Device.Ch[1].Hz_Count:=Device.RX.DI1_Float.tReal;
Device.Ch[2].Hz_Count:=Device.RX.DI2_Float.tReal;
Device.Ch[3].Hz_Count:=Device.RX.DI3_Float.tReal;
Device.Ch[4].Hz_Count:=Device.RX.DI4_Float.tReal;
Device.Ch[5].Hz_Count:=Device.RX.DI5_Float.tReal;
Device.Ch[6].Hz_Count:=Device.RX.DI6_Float.tReal;
Device.Ch[7].Hz_Count:=Device.RX.DI7_Float.tReal;
Device.Ch[8].Hz_Count:=Device.RX.DI8_Float.tReal;

Device.Ch[1].Totaliser:=Device.RX.DI1_Total.tReal;
Device.Ch[2].Totaliser:=Device.RX.DI2_Total.tReal;
Device.Ch[3].Totaliser:=Device.RX.DI3_Total.tReal;
Device.Ch[4].Totaliser:=Device.RX.DI4_Total.tReal;
Device.Ch[5].Totaliser:=Device.RX.DI5_Total.tReal;
Device.Ch[6].Totaliser:=Device.RX.DI6_Total.tReal;
Device.Ch[7].Totaliser:=Device.RX.DI7_Total.tReal;
Device.Ch[8].Totaliser:=Device.RX.DI8_Total.tReal;

Device.Ch[1].Raw:=Device.RX.DI1_DI_8.tByte[1].0;
Device.Ch[2].Raw:=Device.RX.DI1_DI_8.tByte[1].1;
Device.Ch[3].Raw:=Device.RX.DI1_DI_8.tByte[1].2;
Device.Ch[4].Raw:=Device.RX.DI1_DI_8.tByte[1].3;
Device.Ch[5].Raw:=Device.RX.DI1_DI_8.tByte[1].4;
Device.Ch[6].Raw:=Device.RX.DI1_DI_8.tByte[1].5;
Device.Ch[7].Raw:=Device.RX.DI1_DI_8.tByte[1].6;
Device.Ch[8].Raw:=Device.RX.DI1_DI_8.tByte[1].7;





Device.TX.Counter_Reset.8:=Device.Ch[1].Reset_Count;
Device.TX.Totaliser_Reset.8:=Device.Ch[1].Reset_Totaliser;

Device.TX.Counter_Reset.9:=Device.Ch[2].Reset_Count;
Device.TX.Totaliser_Reset.9:=Device.Ch[2].Reset_Totaliser;

Device.TX.Counter_Reset.10:=Device.Ch[3].Reset_Count;
Device.TX.Totaliser_Reset.10:=Device.Ch[3].Reset_Totaliser;

Device.TX.Counter_Reset.11:=Device.Ch[4].Reset_Count;
Device.TX.Totaliser_Reset.11:=Device.Ch[4].Reset_Totaliser;

Device.TX.Counter_Reset.12:=Device.Ch[5].Reset_Count;
Device.TX.Totaliser_Reset.12:=Device.Ch[5].Reset_Totaliser;

Device.TX.Counter_Reset.13:=Device.Ch[6].Reset_Count;
Device.TX.Totaliser_Reset.13:=Device.Ch[6].Reset_Totaliser;

Device.TX.Counter_Reset.14:=Device.Ch[7].Reset_Count;
Device.TX.Totaliser_Reset.14:=Device.Ch[7].Reset_Totaliser;

Device.TX.Counter_Reset.15:=Device.Ch[8].Reset_Count;
Device.TX.Totaliser_Reset.15:=Device.Ch[8].Reset_Totaliser;

END_FUNCTION

// Level_1/Analog_Pump_HMI_Sync
FUNCTION_BLOCK Analog_Pump_HMI_Sync
VAR_INPUT
	Sync:BOOL;
END_VAR
VAR_OUTPUT
	StrStatus:STRING;
	StrMode:String;
END_VAR
VAR
	Buffer:cAnalog_Pump;
	R_Trig_0: R_trig;
	Sync_1: BOOL;
	Sync_2: BOOL;
	PLC_Changes:UINT;
	HMI_Changes:UINT;
	
END_VAR

VAR_IN_OUT
	HMI:cAnalog_Pump;
	Local:cAnalog_Pump;
END_VAR

(* body of a kind this reader does not render *)

END_FUNCTION_BLOCK

// Level_1/Contactor_HMI_Sync_UDFB
FUNCTION_BLOCK Contactor_HMI_Sync_UDFB
VAR_INPUT
	Sync:BOOL;
END_VAR
VAR_OUTPUT
	strMode:STRING;
	strStatus:STRING;
END_VAR
VAR
	Buffer:Burkert.Contactor_DUT;
	R_Trig_0: R_trig;
	Sync_1: BOOL;
	Sync_2: BOOL;
	PLC_Changes:UINT;
	HMI_Changes:UINT;
	
END_VAR

VAR_IN_OUT
	HMI:Burkert.Contactor_DUT;
	Local:Burkert.Contactor_DUT;
END_VAR

(* body of a kind this reader does not render *)

END_FUNCTION_BLOCK

// Level_1/Eaton_VFD_HMI_Sync
FUNCTION_BLOCK Eaton_VFD_HMI_Sync
VAR_INPUT
	Sync:BOOL;
END_VAR
VAR_OUTPUT
	StrStatus:STRING;
	StrMode:String;
END_VAR
VAR
	Buffer:cVFD_Eaton_DUT;
	R_Trig_0: R_trig;
	Sync_1: BOOL;
	Sync_2: BOOL;
	PLC_Changes:UINT;
	HMI_Changes:UINT;
	
END_VAR

VAR_IN_OUT
	HMI:cVFD_Eaton_DUT;
	Local:cVFD_Eaton_DUT;
END_VAR

(* body of a kind this reader does not render *)

END_FUNCTION_BLOCK

// Level_1/M_Pump_HMI_Sync
FUNCTION_BLOCK M_Pump_HMI_Sync
VAR_INPUT
	Sync:BOOL;
END_VAR
VAR_OUTPUT
	StrStatus:STRING;
	StrMode:String;
END_VAR
VAR
	Buffer:cM_Pump;
	R_Trig_0: R_trig;
	Sync_1: BOOL;
	Sync_2: BOOL;
	PLC_Changes:UINT;
	HMI_Changes:UINT;
	
END_VAR

VAR_IN_OUT
	HMI:cM_Pump;
	Local:cM_Pump;
END_VAR

(* body of a kind this reader does not render *)

END_FUNCTION_BLOCK

// Level_2/PID_HMI_Sync_UDFB
FUNCTION_BLOCK PID_HMI_Sync_UDFB
VAR_INPUT
	Sync:BOOL;
END_VAR
VAR_OUTPUT
	strMode:STRING;
	strStatus:STRING;
END_VAR
VAR
	Buffer:cPID_DUT;
	R_Trig_0: R_trig;
	Sync_1: BOOL;
	Sync_2: BOOL;
	PLC_Changes:UINT;
	HMI_Changes:UINT;
	
END_VAR

VAR_IN_OUT
	HMI:cPID_DUT;
	Local:cPID_DUT;
END_VAR

(* body of a kind this reader does not render *)

END_FUNCTION_BLOCK

// Level_3/Brite_HMI_Sync
FUNCTION_BLOCK Brite_HMI_Sync
VAR_INPUT
	Sync:BOOL;
END_VAR
VAR_OUTPUT
END_VAR
VAR
	Buffer:cBrite_DUT;
	R_Trig_0: R_trig;
	Sync_1: BOOL;
	Sync_2: BOOL;
	PLC_Changes:UINT;
	HMI_Changes:UINT;
	
	//PID_0: PID_HMI_Sync_UDFB;
	PID_Match: BOOL;
	Status_Match: BOOL;
	PID_Coompare: UINT;
	Status_Compare: UINT;
END_VAR

VAR_IN_OUT
	HMI:cBrite_DUT;
	Local:cBrite_DUT;
END_VAR

(* body of a kind this reader does not render *)

END_FUNCTION_BLOCK

// Level_3/Fermenter_HMI_Sync
FUNCTION_BLOCK Fermenter_HMI_Sync
VAR_INPUT
	Sync:BOOL;
END_VAR
VAR_OUTPUT
END_VAR
VAR
	Buffer:cFermenter_DUT;
	R_Trig_0: R_trig;
	Sync_1: BOOL;
	Sync_2: BOOL;
	PLC_Changes:UINT;
	HMI_Changes:UINT;
	
	//PID_0: PID_HMI_Sync_UDFB;
	PID_Match: BOOL;
	Status_Match: BOOL;
	PID_Coompare: UINT;
	Status_Compare: UINT;
END_VAR

VAR_IN_OUT
	HMI:cFermenter_DUT;
	Local:cFermenter_DUT;
END_VAR

(* body of a kind this reader does not render *)

END_FUNCTION_BLOCK

// Adam_6050_FB
FUNCTION Adam_6050_FB : BOOL
VAR_INPUT
	HSC_0_Enable:BOOL:=FALSE;
	HSC_0_Reset:BOOL:=FALSE;
	HSC_1_Enable:BOOL:=FALSE;
	HSC_1_Reset:BOOL:=FALSE;
	HSC_2_Enable:BOOL:=FALSE;
	HSC_2_Reset:BOOL:=FALSE;
	HSC_3_Enable:BOOL:=FALSE;
	HSC_3_Reset:BOOL:=FALSE;
	HSC_4_Enable:BOOL:=FALSE;
	HSC_4_Reset:BOOL:=FALSE;
	HSC_5_Enable:BOOL:=FALSE;
	HSC_5_Reset:BOOL:=FALSE;
	HSC_6_Enable:BOOL:=FALSE;
	HSC_6_Reset:BOOL:=FALSE;
	HSC_7_Enable:BOOL:=FALSE;
	HSC_7_Reset:BOOL:=FALSE;
	HSC_8_Enable:BOOL:=FALSE;
	HSC_8_Reset:BOOL:=FALSE;
	HSC_9_Enable:BOOL:=FALSE;
	HSC_9_Reset:BOOL:=FALSE;
	HSC_10_Enable:BOOL:=FALSE;
	HSC_10_Reset:BOOL:=FALSE;
	HSC_11_Enable:BOOL:=FALSE;
	HSC_11_Reset:BOOL:=FALSE;
	
	DO_0:BOOL:=FALSE;
	DO_1:BOOL:=FALSE;
	DO_2:BOOL:=FALSE;
	DO_3:BOOL:=FALSE;
	DO_4:BOOL:=FALSE;
	DO_5:BOOL:=FALSE;
//	DO_6:BOOL;
//	DO_7:BOOL;
	RX_DI_4x300: WORD;
	RX_Counts_4x0: ARRAY[0..11] OF UDINT;
END_VAR
VAR_OUTPUT
	HSC_0:UDINT;
	HSC_1:UDINT;
	HSC_2:UDINT;
	HSC_3:UDINT;
	HSC_4:UDINT;
	HSC_5:UDINT;
	HSC_6:UDINT;
	HSC_7:UDINT;
	HSC_8:UDINT;
	HSC_9:UDINT;
	HSC_10:UDINT;
	HSC_11:UDINT;
	
	DI_0:BOOL;
	DI_1:BOOL;
	DI_2:BOOL;
	DI_3:BOOL;
	DI_4:BOOL;
	DI_5:BOOL;
	DI_6:BOOL;
	DI_7:BOOL;
	DI_8:BOOL;
	DI_9:BOOL;
	DI_10:BOOL;
	DI_11:BOOL;
	
	

	
	
	TX_DO_4x302: WORD;
	TX_Counts_Control_0x32: ARRAY[0..2] OF WORD;
END_VAR
VAR
END_VAR

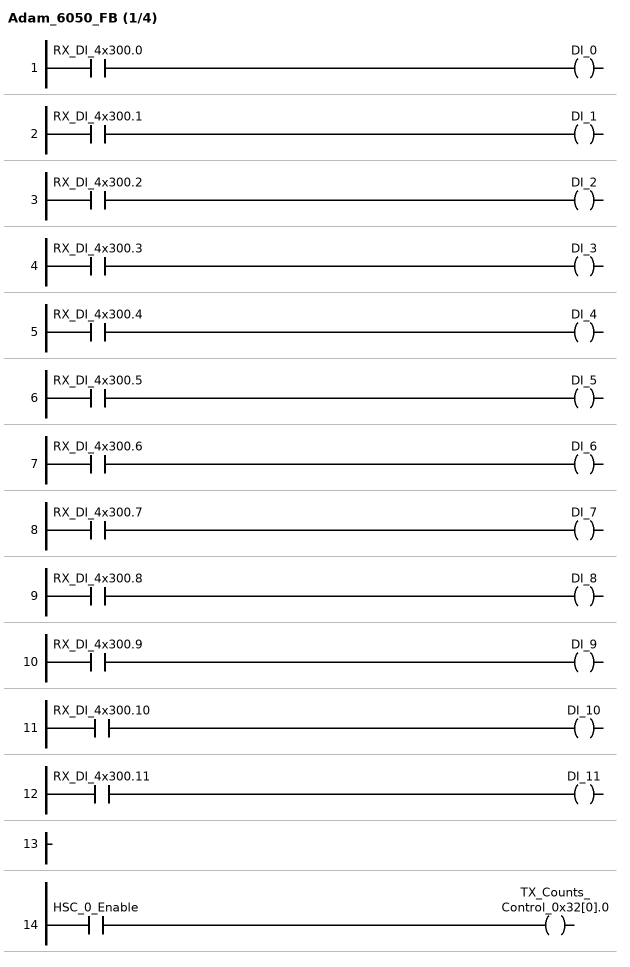
// NETWORK 1
DI_0 := RX_DI_4x300.0;

// NETWORK 2
DI_1 := RX_DI_4x300.1;

// NETWORK 3
DI_2 := RX_DI_4x300.2;

// NETWORK 4
DI_3 := RX_DI_4x300.3;

// NETWORK 5
DI_4 := RX_DI_4x300.4;

// NETWORK 6
DI_5 := RX_DI_4x300.5;

// NETWORK 7
DI_6 := RX_DI_4x300.6;

// NETWORK 8
DI_7 := RX_DI_4x300.7;

// NETWORK 9
DI_8 := RX_DI_4x300.8;

// NETWORK 10
DI_9 := RX_DI_4x300.9;

// NETWORK 11
DI_10 := RX_DI_4x300.10;

// NETWORK 12
DI_11 := RX_DI_4x300.11;

// NETWORK 13

// NETWORK 14
TX_Counts_Control_0x32[0].0 := HSC_0_Enable;

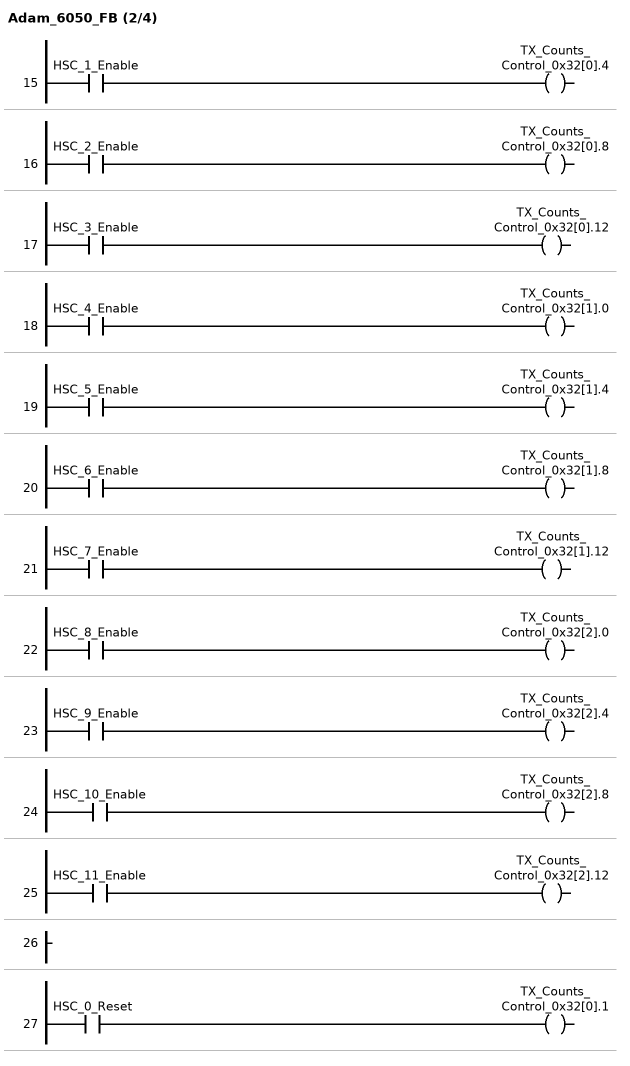
// NETWORK 15
TX_Counts_Control_0x32[0].4 := HSC_1_Enable;

// NETWORK 16
TX_Counts_Control_0x32[0].8 := HSC_2_Enable;

// NETWORK 17
TX_Counts_Control_0x32[0].12 := HSC_3_Enable;

// NETWORK 18
TX_Counts_Control_0x32[1].0 := HSC_4_Enable;

// NETWORK 19
TX_Counts_Control_0x32[1].4 := HSC_5_Enable;

// NETWORK 20
TX_Counts_Control_0x32[1].8 := HSC_6_Enable;

// NETWORK 21
TX_Counts_Control_0x32[1].12 := HSC_7_Enable;

// NETWORK 22
TX_Counts_Control_0x32[2].0 := HSC_8_Enable;

// NETWORK 23
TX_Counts_Control_0x32[2].4 := HSC_9_Enable;

// NETWORK 24
TX_Counts_Control_0x32[2].8 := HSC_10_Enable;

// NETWORK 25
TX_Counts_Control_0x32[2].12 := HSC_11_Enable;

// NETWORK 26

// NETWORK 27
TX_Counts_Control_0x32[0].1 := HSC_0_Reset;

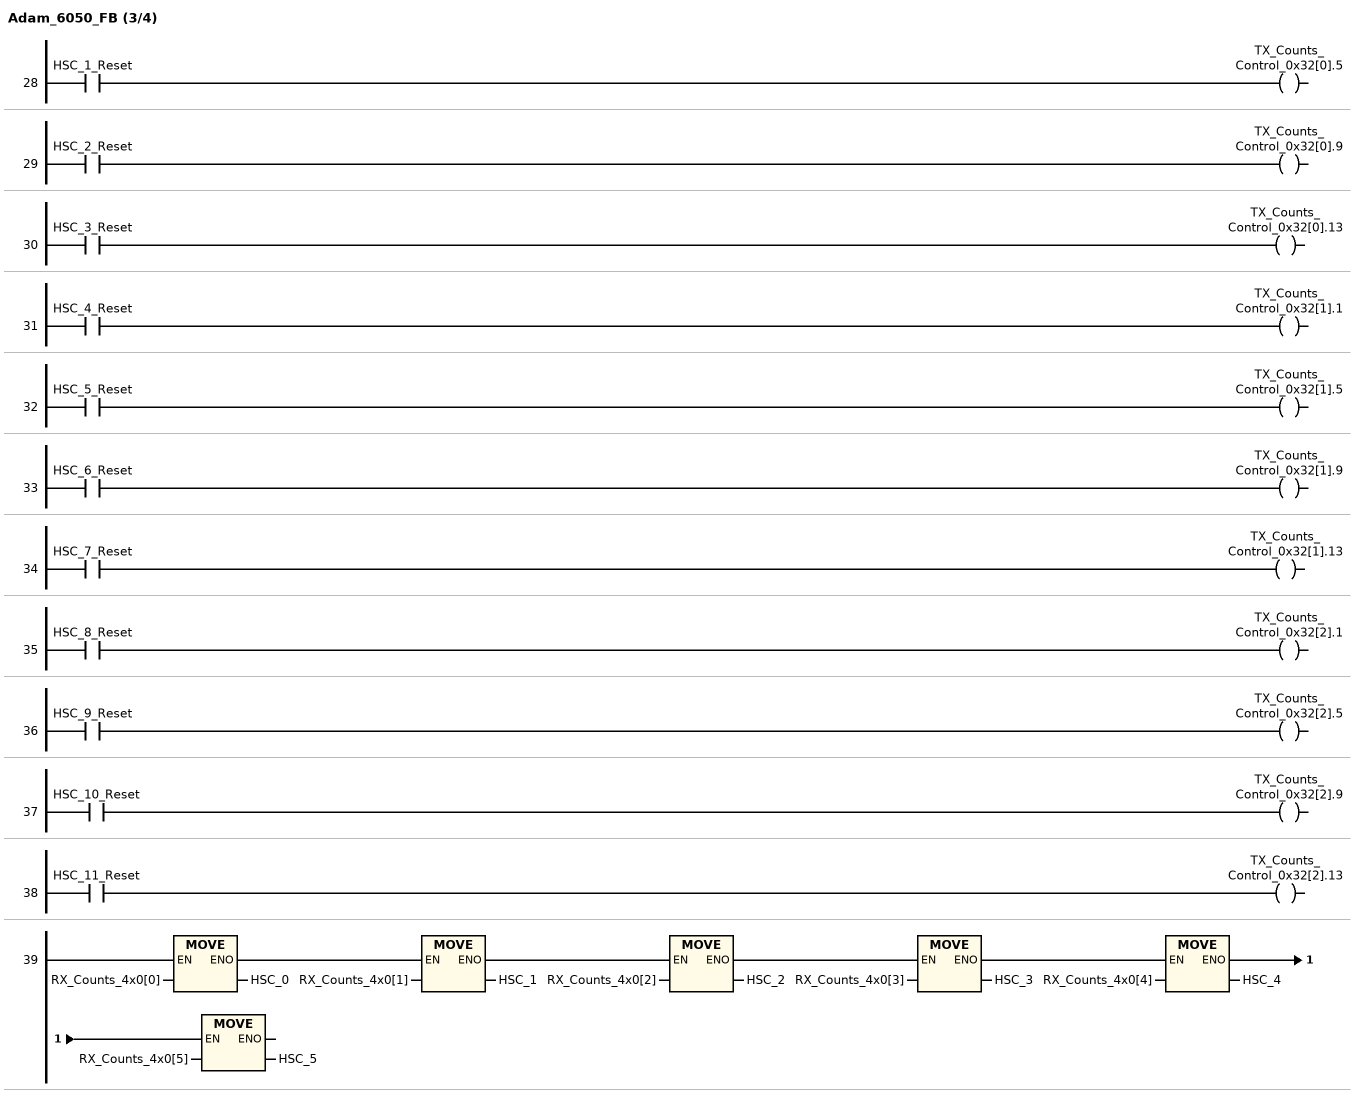
// NETWORK 28
TX_Counts_Control_0x32[0].5 := HSC_1_Reset;

// NETWORK 29
TX_Counts_Control_0x32[0].9 := HSC_2_Reset;

// NETWORK 30
TX_Counts_Control_0x32[0].13 := HSC_3_Reset;

// NETWORK 31
TX_Counts_Control_0x32[1].1 := HSC_4_Reset;

// NETWORK 32
TX_Counts_Control_0x32[1].5 := HSC_5_Reset;

// NETWORK 33
TX_Counts_Control_0x32[1].9 := HSC_6_Reset;

// NETWORK 34
TX_Counts_Control_0x32[1].13 := HSC_7_Reset;

// NETWORK 35
TX_Counts_Control_0x32[2].1 := HSC_8_Reset;

// NETWORK 36
TX_Counts_Control_0x32[2].5 := HSC_9_Reset;

// NETWORK 37
TX_Counts_Control_0x32[2].9 := HSC_10_Reset;

// NETWORK 38
TX_Counts_Control_0x32[2].13 := HSC_11_Reset;

// NETWORK 39
HSC_0 := RX_Counts_4x0[0];
HSC_1 := RX_Counts_4x0[1];
HSC_2 := RX_Counts_4x0[2];
HSC_3 := RX_Counts_4x0[3];
HSC_4 := RX_Counts_4x0[4];
HSC_5 := RX_Counts_4x0[5];

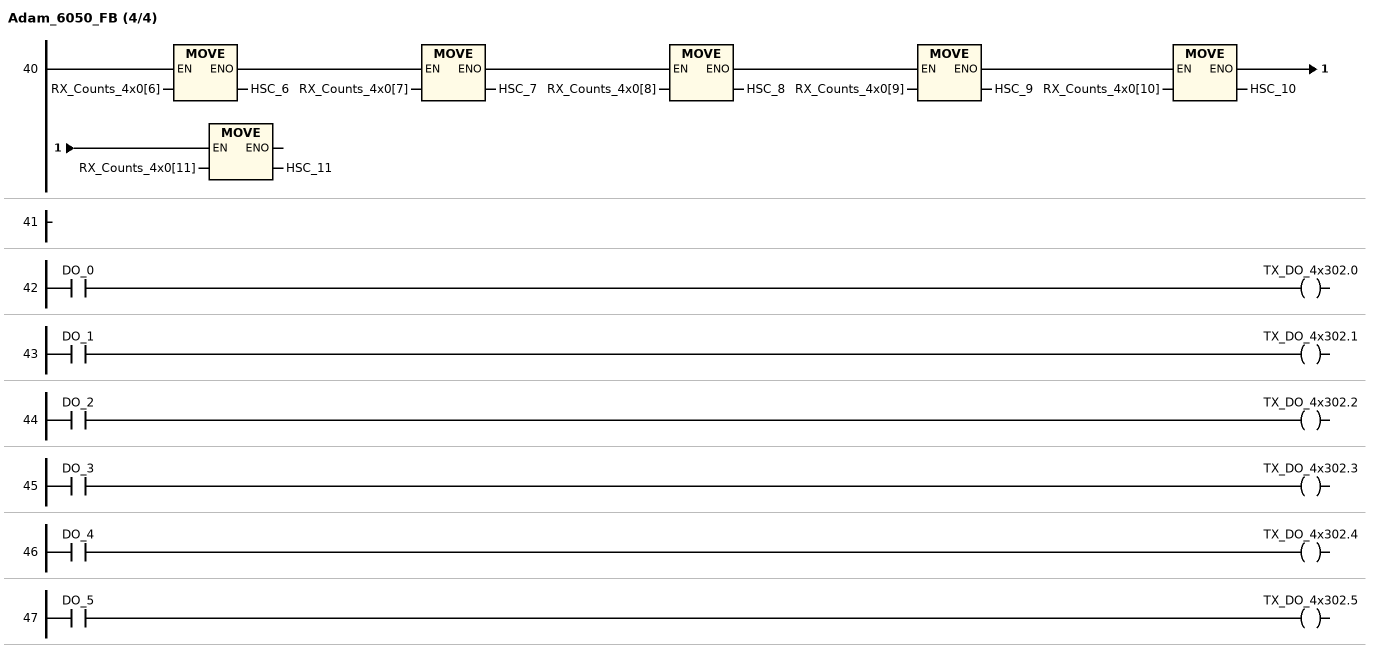
// NETWORK 40
HSC_6 := RX_Counts_4x0[6];
HSC_7 := RX_Counts_4x0[7];
HSC_8 := RX_Counts_4x0[8];
HSC_9 := RX_Counts_4x0[9];
HSC_10 := RX_Counts_4x0[10];
HSC_11 := RX_Counts_4x0[11];

// NETWORK 41

// NETWORK 42
TX_DO_4x302.0 := DO_0;

// NETWORK 43
TX_DO_4x302.1 := DO_1;

// NETWORK 44
TX_DO_4x302.2 := DO_2;

// NETWORK 45
TX_DO_4x302.3 := DO_3;

// NETWORK 46
TX_DO_4x302.4 := DO_4;

// NETWORK 47
TX_DO_4x302.5 := DO_5;

END_FUNCTION

// Adam_6250
FUNCTION Adam_6250 : bool
VAR_INPUT
	Device:REFERENCE TO cAdam_6250;
END_VAR

VAR
END_VAR

Device.DI[0].DI:=Device.Rx_DI.0;
Device.DI[1].DI:=Device.Rx_DI.1;
Device.DI[2].DI:=Device.Rx_DI.2;
Device.DI[3].DI:=Device.Rx_DI.3;
Device.DI[4].DI:=Device.Rx_DI.4;
Device.DI[5].DI:=Device.Rx_DI.5;
Device.DI[6].DI:=Device.Rx_DI.6;
Device.DI[7].DI:=Device.Rx_DI.7;

Device.DI[0].Count:=Device.RX_Counter_Values[0];
Device.DI[1].Count:=Device.RX_Counter_Values[1];
Device.DI[2].Count:=Device.RX_Counter_Values[2];
Device.DI[3].Count:=Device.RX_Counter_Values[3];
Device.DI[4].Count:=Device.RX_Counter_Values[4];
Device.DI[5].Count:=Device.RX_Counter_Values[5];
Device.DI[6].Count:=Device.RX_Counter_Values[6];
Device.DI[7].Count:=Device.RX_Counter_Values[7];

Device.DI[0].Frequency:=TO_REAL(Device.RX_Counter_Values[0])/10;
Device.DI[1].Frequency:=TO_REAL(Device.RX_Counter_Values[1])/10;
Device.DI[2].Frequency:=TO_REAL(Device.RX_Counter_Values[2])/10;
Device.DI[3].Frequency:=TO_REAL(Device.RX_Counter_Values[3])/10;
Device.DI[4].Frequency:=TO_REAL(Device.RX_Counter_Values[4])/10;
Device.DI[5].Frequency:=TO_REAL(Device.RX_Counter_Values[5])/10;
Device.DI[6].Frequency:=TO_REAL(Device.RX_Counter_Values[6])/10;
Device.DI[7].Frequency:=TO_REAL(Device.RX_Counter_Values[7])/10;

Device.Tx_Counter_Control[0].0:=Device.DI[0].Enable_HSC;
Device.Tx_Counter_Control[0].1:=Device.DI[1].Enable_HSC;
Device.Tx_Counter_Control[0].2:=Device.DI[2].Enable_HSC;
Device.Tx_Counter_Control[0].3:=Device.DI[3].Enable_HSC;
Device.Tx_Counter_Control[0].4:=Device.DI[4].Enable_HSC;
Device.Tx_Counter_Control[0].5:=Device.DI[5].Enable_HSC;
Device.Tx_Counter_Control[0].6:=Device.DI[6].Enable_HSC;
Device.Tx_Counter_Control[0].7:=Device.DI[7].Enable_HSC;

Device.Tx_Counter_Control[1].0:=Device.DI[0].Clear_HSC;
Device.Tx_Counter_Control[1].1:=Device.DI[1].Clear_HSC;
Device.Tx_Counter_Control[1].2:=Device.DI[2].Clear_HSC;
Device.Tx_Counter_Control[1].3:=Device.DI[3].Clear_HSC;
Device.Tx_Counter_Control[1].4:=Device.DI[4].Clear_HSC;
Device.Tx_Counter_Control[1].5:=Device.DI[5].Clear_HSC;
Device.Tx_Counter_Control[1].6:=Device.DI[6].Clear_HSC;
Device.Tx_Counter_Control[1].7:=Device.DI[7].Clear_HSC;

Device.Tx_Counter_Control[2].0:=Device.DI[0].Clear_Overflow;
Device.Tx_Counter_Control[2].1:=Device.DI[1].Clear_Overflow;
Device.Tx_Counter_Control[2].2:=Device.DI[2].Clear_Overflow;
Device.Tx_Counter_Control[2].3:=Device.DI[3].Clear_Overflow;
Device.Tx_Counter_Control[2].4:=Device.DI[4].Clear_Overflow;
Device.Tx_Counter_Control[2].5:=Device.DI[5].Clear_Overflow;
Device.Tx_Counter_Control[2].6:=Device.DI[6].Clear_Overflow;
Device.Tx_Counter_Control[2].7:=Device.DI[7].Clear_Overflow;

Device.Tx_DO.0	:=device.Dout[0].Dout;
Device.Tx_DO.1	:=device.Dout[1].Dout;
Device.Tx_DO.2	:=device.Dout[2].Dout;
Device.Tx_DO.3	:=device.Dout[3].Dout;
Device.Tx_DO.4	:=device.Dout[4].Dout;
Device.Tx_DO.5	:=device.Dout[5].Dout;
Device.Tx_DO.6	:=device.Dout[6].Dout;

Device.Tx_Pulse_Width_Low[0] :=Device.Dout[0].Pulse_Output_Low_Width;
Device.Tx_Pulse_Width_Low[1] :=Device.Dout[1].Pulse_Output_Low_Width;
Device.Tx_Pulse_Width_Low[2] :=Device.Dout[2].Pulse_Output_Low_Width;
Device.Tx_Pulse_Width_Low[3] :=Device.Dout[3].Pulse_Output_Low_Width;
Device.Tx_Pulse_Width_Low[4] :=Device.Dout[4].Pulse_Output_Low_Width;
Device.Tx_Pulse_Width_Low[5] :=Device.Dout[5].Pulse_Output_Low_Width;
Device.Tx_Pulse_Width_Low[6] :=Device.Dout[6].Pulse_Output_Low_Width;

Device.Tx_Pulse_Width_High[0]	:=Device.Dout[0].Pulse_Output_High_Width;
Device.Tx_Pulse_Width_High[1]	:=Device.Dout[1].Pulse_Output_High_Width;
Device.Tx_Pulse_Width_High[2]	:=Device.Dout[2].Pulse_Output_High_Width;
Device.Tx_Pulse_Width_High[3]	:=Device.Dout[3].Pulse_Output_High_Width;
Device.Tx_Pulse_Width_High[4]	:=Device.Dout[4].Pulse_Output_High_Width;
Device.Tx_Pulse_Width_High[5]	:=Device.Dout[5].Pulse_Output_High_Width;
Device.Tx_Pulse_Width_High[6]	:=Device.Dout[6].Pulse_Output_High_Width;

Device.Tx_Set_Absolute_Pulse[0]	:=Device.Dout[0].Set_Absolute_Pulse;
Device.Tx_Set_Absolute_Pulse[1]	:=Device.Dout[1].Set_Absolute_Pulse;
Device.Tx_Set_Absolute_Pulse[2]	:=Device.Dout[2].Set_Absolute_Pulse;
Device.Tx_Set_Absolute_Pulse[3]	:=Device.Dout[3].Set_Absolute_Pulse;
Device.Tx_Set_Absolute_Pulse[4]	:=Device.Dout[4].Set_Absolute_Pulse;
Device.Tx_Set_Absolute_Pulse[5]	:=Device.Dout[5].Set_Absolute_Pulse;
Device.Tx_Set_Absolute_Pulse[6]	:=Device.Dout[6].Set_Absolute_Pulse;

Device.Tx_Set_Incremental_Pulse[0]	:=Device.Dout[0].Set_Incremental_Pulse;
Device.Tx_Set_Incremental_Pulse[1]	:=Device.Dout[1].Set_Incremental_Pulse;
Device.Tx_Set_Incremental_Pulse[2]	:=Device.Dout[2].Set_Incremental_Pulse;
Device.Tx_Set_Incremental_Pulse[3]	:=Device.Dout[3].Set_Incremental_Pulse;
Device.Tx_Set_Incremental_Pulse[4]	:=Device.Dout[4].Set_Incremental_Pulse;
Device.Tx_Set_Incremental_Pulse[5]	:=Device.Dout[5].Set_Incremental_Pulse;
Device.Tx_Set_Incremental_Pulse[6]	:=Device.Dout[6].Set_Incremental_Pulse;

END_FUNCTION

// Level_0_Remote_IO/MicroControl/MC4AI
FUNCTION MC4AI 
VAR_INPUT
	GW_TCP_State:ModbusTCPComState;
END_VAR

VAR
END_VAR


VAR_IN_OUT
	GW:MicroControl_4AI;
END_VAR

GW.GW_TCP_State:=GW_TCP_State;

IF NOT(GW_TCP_State=10) THEN
	GW.PV[0]:= (TO_REAL(GW.PV_RX[0])/1000);
	GW.PV[1]:= (TO_REAL(GW.PV_RX[1])/1000);
	GW.PV[2]:= (TO_REAL(GW.PV_RX[2])/1000);
	GW.PV[3]:= (TO_REAL(GW.PV_RX[3])/1000);
ELSE
	GW.PV[0]:=(-9999999);
	GW.PV[1]:=(-9999999);
	GW.PV[2]:=(-9999999);
	GW.PV[3]:=(-9999999);
END_IF;

END_FUNCTION

// MB0_RTD
FUNCTION_BLOCK MB0_RTD
VAR_INPUT
	Online:BOOL;
	Device: REFERENCE TO cMB0_RTD;
	
	CH1: REFERENCE TO 	Burkert.cAIT;
	CH1_Probe_Type:		eMB0_RTD_Input_Type;
	CH2: REFERENCE TO 	Burkert.cAIT;
	CH2_Probe_Type:		eMB0_RTD_Input_Type;
	CH3: REFERENCE TO 	Burkert.cAIT;
	CH3_Probe_Type:		eMB0_RTD_Input_Type;
	CH4: REFERENCE TO 	Burkert.cAIT;
	CH4_Probe_Type:		eMB0_RTD_Input_Type;
	System_Units:eUnits;
END_VAR
VAR_OUTPUT
END_VAR
VAR
	Alarm:ARRAY[0..3] OF Burkert.Analog_Alarm_UDFB;
END_VAR

CASE System_Units OF
	eUnits.C:
		Device.TX.Holding_1218[0]:=eMB0_RTD_Units.C;
		Device.TX.Holding_1218[1]:=eMB0_RTD_Units.C;
		Device.TX.Holding_1218[2]:=eMB0_RTD_Units.C;
		Device.TX.Holding_1218[3]:=eMB0_RTD_Units.C;
	eUnits.F:
		Device.TX.Holding_1218[0]:=eMB0_RTD_Units.F;
		Device.TX.Holding_1218[1]:=eMB0_RTD_Units.F;
		Device.TX.Holding_1218[2]:=eMB0_RTD_Units.F;
		Device.TX.Holding_1218[3]:=eMB0_RTD_Units.F;
	eUnits.K:
		Device.TX.Holding_1218[0]:=eMB0_RTD_Units.k;
		Device.TX.Holding_1218[1]:=eMB0_RTD_Units.k;
		Device.TX.Holding_1218[2]:=eMB0_RTD_Units.k;
		Device.TX.Holding_1218[3]:=eMB0_RTD_Units.k;
END_CASE

Device.TX.Holding_31[0]:=CH1_Probe_Type;
Device.TX.Holding_31[1]:=CH1_Probe_Type;
Device.TX.Holding_31[2]:=CH1_Probe_Type;
Device.TX.Holding_31[3]:=CH1_Probe_Type;


CH1.Sensor.EU:=TO_REAL(Device.RX.Holding_41[0])/10;
CH2.Sensor.EU:=TO_REAL(Device.RX.Holding_41[1])/10;
CH3.Sensor.EU:=TO_REAL(Device.RX.Holding_41[2])/10;
CH4.Sensor.EU:=TO_REAL(Device.RX.Holding_41[3])/10;

Alarm[0](
	Config:=CH1.Sensor.Alarm_Config,
	EU:=CH1.Sensor.EU,
	Debounce_Active:=CH1.Sensor.Alarm_Config.Silence, 
	Status =>CH1.Sensor.Status.eStatus,
	Percent_Alarm=>CH1.Sensor.Alarm_Config.PCT_Alarm
	);
Alarm[1](
	Config:=CH2.Sensor.Alarm_Config,
	EU:=CH2.Sensor.EU,
	Debounce_Active:=CH2.Sensor.Alarm_Config.Silence, 
	Status =>CH2.Sensor.Status.eStatus,
	Percent_Alarm=>CH2.Sensor.Alarm_Config.PCT_Alarm
	);
Alarm[2](
	Config:=CH3.Sensor.Alarm_Config,
	EU:=CH3.Sensor.EU,
	Debounce_Active:=CH3.Sensor.Alarm_Config.Silence, 
	Status =>CH3.Sensor.Status.eStatus,
	Percent_Alarm=>CH3.Sensor.Alarm_Config.PCT_Alarm
	);
Alarm[3](
	Config:=CH4.Sensor.Alarm_Config,
	EU:=CH4.Sensor.EU,
	Debounce_Active:=CH4.Sensor.Alarm_Config.Silence, 
	Status =>CH4.Sensor.Status.eStatus,
	Percent_Alarm=>CH4.Sensor.Alarm_Config.PCT_Alarm
	);
	
IF NOT(Online) THEN
	CH1.Sensor.Status.eStatus:=Burkert.eSensor_Status.Offline;
	CH2.Sensor.Status.eStatus:=Burkert.eSensor_Status.Offline;
	CH3.Sensor.Status.eStatus:=Burkert.eSensor_Status.Offline;
	CH4.Sensor.Status.eStatus:=Burkert.eSensor_Status.Offline;
END_IF

END_FUNCTION_BLOCK

// Level_1_Devices/Burkert Library/Analog_Alarm_UDFB
FUNCTION_BLOCK Analog_Alarm_UDFB
VAR_INPUT
	Config	:	REFERENCE TO Burkert.cAlarm_Config;
	EU:REAL  ;
	Debounce_Active:BOOL;
	
END_VAR
VAR_OUTPUT
	Status:eSensor_Status;
	Percent_Alarm:REAL;
	
END_VAR
VAR
	ALARM: BURKERT_OSCAT_BASIC.ALARM_2;
	Warn_Debounce: TON;
	Alarm_Debounce: TON;
	ALarm_PCT:ARRAY[0..4] OF REAL;
	
END_VAR

Status:=run();

METHOD run : eSensor_Status
VAR_INPUT

END_VAR

VAR_OUTPUT

END_VAR
(* body of a kind this reader does not render *)
END_METHOD

END_FUNCTION_BLOCK

// SIO_MB12CDR
FUNCTION_BLOCK SIO_MB12CDR
VAR_INPUT
	Online:BOOL;
	Device : REFERENCE TO cSIO_MB12CDR;
	FIT_0:REFERENCE TO Burkert.cBase_FIT;
	FIT_1:REFERENCE TO Burkert.cBase_FIT;
	FIT_2:REFERENCE TO	Burkert.cBase_FIT;
	FIT_3:REFERENCE TO Burkert.cBase_FIT;
END_VAR
VAR_OUTPUT
END_VAR
VAR
END_VAR

END_FUNCTION_BLOCK

// Contactor
FUNCTION_BLOCK Contactor
VAR_INPUT
	NO_OL:BOOL;
	NO_FWD_Aux:BOOL;
	NO_REV_Aux:BOOL;


	Allow_Reverse:BOOL;
	Inhibit_FWD:BOOL:=FALSE;
	Inhibit_Rev:BOOL:=FALSE;
	Bump_Duration:TIME:=T#1S;
END_VAR

VAR_IN_OUT
	Contactor:cContactor;
END_VAR

VAR_OUTPUT
	Q_FWD:BOOL;
	Q_REV:Bool;
END_VAR


VAR
	local_FWD:BOOL;
	Local_Rev:BOOL;
	Bump_Timer:TP;
	Engage_Ton:TON;
	
END_VAR

Bump_Timer(
	PT:=Bump_Duration, 
	IN:= (Contactor.Mode.eMode=Contactor_modes.Bump_FWD OR Contactor.Mode.eMode=Contactor_modes.Bump_rev)
);
	

Engage_Ton(PT:=T#1S, IN:=(Q_FWD OR Q_REV));

CASE Contactor.Mode.eMode OF
	Contactor_modes.Disabled:
		Local_FWD:=FALSE;
		Local_Rev:=FALSE;
	Contactor_modes.Auto:
		Local_FWD:=Contactor.PLC_CMD_FWD;
		Local_Rev:=Contactor.PLC_CMD_Rev;
	Contactor_modes.Bump_FWD:
		Local_FWD:=Bump_Timer.Q;
		Local_REV:=FALSE;
	Contactor_modes.Bump_REV:
		Local_FWD:=FALSE;
		Local_REV:=Bump_Timer.Q;
	Contactor_modes.Fwd:
		Local_FWD:=TRUE;
		Local_Rev:=FALSE;
	Contactor_modes.Rev:
		Local_FWD:=FALSE;
		Local_Rev:=TRUE;
END_CASE

//IF Inhibit_FWD THEN local_FWD:=FALSE; END_IF;
//IF Inhibit_Rev THEN Local_REv:=FALSE;	END_IF;
IF NO_OL	THEN 
	Local_FWD:=FALSE;
	Local_Rev:=FALSE;
END_IF;

IF (Local_FWD AND Local_REV) THEN
	Local_FWD:=FALSE;
	Local_Rev:=FALSE;
END_IF;

Q_FWD:=Local_FWD AND NOT(Inhibit_FWD);
Q_Rev:=Local_Rev AND NOT(Inhibit_Rev);

Status();

ACTION Status:
Contactor.Ready :=(
	Contactor.Mode.eMode=Contactor_modes.Auto AND
	NOT(NO_OL)
);

Contactor.Status.eStatus:=eContactor_Status.Idle;
IF Contactor.Mode.eMode=Contactor_modes.Disabled THEN	Contactor.Status.eStatus:=eContactor_Status.Disabled; END_IF;




IF Contactor.Mode.eMode=Contactor_modes.Auto AND Contactor.PLC_CMD_FWD THEN Contactor.Status.eStatus:=eContactor_Status.Auto_FWD; END_IF;
IF Contactor.Mode.eMode=Contactor_modes.Auto AND Contactor.PLC_CMD_REV THEN Contactor.Status.eStatus:=eContactor_Status.Auto_Rev; END_IF;

IF Contactor.Mode.eMode=Contactor_modes.Bump_FWD AND Bump_Timer.Q THEN Contactor.Status.eStatus:=eContactor_Status.Manual_FWD; END_IF;
IF Contactor.Mode.eMode=Contactor_modes.Bump_Rev AND Bump_Timer.Q THEN Contactor.Status.eStatus:=eContactor_Status.Manual_REV; END_IF;

IF Contactor.Mode.eMode=Contactor_modes.Fwd  THEN Contactor.Status.eStatus:=eContactor_Status.Manual_FWD; END_IF;
IF Contactor.Mode.eMode=Contactor_modes.rev  THEN Contactor.Status.eStatus:=eContactor_Status.Manual_REV; END_IF;


IF Local_FWD AND NO_FWD_Aux THEN	Contactor.Status.eStatus:=eContactor_Status.FWD_Limit; END_IF;
IF Local_Rev AND NO_Rev_Aux THEN	Contactor.Status.eStatus:=eContactor_Status.Rev_Limit; END_IF;

IF Engage_Ton.Q AND NOT(NO_FWD_Aux OR NO_REV_Aux) THEN Contactor.Status.eStatus:=eContactor_Status.Failed_to_Engange; END_IF;
IF NO_OL THEN Contactor.Status.eStatus:=eContactor_Status.Tripped; END_IF;
END_ACTION

END_FUNCTION_BLOCK

// Contactor_Control_UDFB
FUNCTION_BLOCK Contactor_Control_UDFB
VAR_INPUT
	//Interlock_NC:BOOL;
	//Permissive_NC:BOOL;
	
	Allow_Reverse:BOOL;
	Inhibit_FWD:BOOL:=FALSE;
	Inhibit_Rev:BOOL:=FALSE;
	Bump_Duration:TIME:=T#1S;
END_VAR
VAR_OUTPUT
	Q_FWD:BOOL;
	Q_REV:Bool;
END_VAR
VAR
	//F_TRIG_0: F_trig;
	TP_0: TP;
	F_TRIG_1: F_trig;
	TP_1: TP;
END_VAR
VAR_IN_OUT
	Contactor:cContactor;
END_VAR
VAR // added by the converter: edge detectors and wires of the graphical bodies
    _w1, _w2, _w4, _w5, _w6, _w7, _w8, _w10, _w11, _w12 : BOOL;
    _w3, _w9 : ANY;
END_VAR

_w1 := Contactor.Mode.eMode = Contactor_Modes.Auto;
_w2 := _w1 AND Contactor.PLC_CMD_FWD;
_w3 := SEL(_w2, eContactor_Status.OFF, eContactor_Status.Auto_FWD);
_w4 := Contactor.Mode.eMode = Contactor_Modes.Fwd;
TP_1(IN := Contactor.Mode.eMode = Contactor_Modes.Bump_FWD, PT := Bump_Duration); // TP
_w5 := _w4 OR TP_1.Q;
_w6 := _w2 OR _w5;
_w7 := _w6 AND NOT Inhibit_FWD AND NOT (Contactor.Mode.eMode=Contactor_Modes.Disabled);
Contactor.Q1 := _w7;
Q_FWD := _w7;
_w8 := _w1 AND Contactor.PLC_CMD_Rev;
_w9 := SEL(_w8, SEL((_w2 OR _w5) AND Inhibit_FWD, SEL(_w5, _w3, eContactor_Status.Manual_FWD), eContactor_Status.FWD_Limit), eContactor_Status.Auto_Rev);
_w10 := Contactor.Mode.eMode = Contactor_Modes.Rev;
TP_0(IN := Contactor.Mode.eMode = Contactor_Modes.Bump_REV, PT := Bump_Duration); // TP
_w11 := _w10 OR TP_0.Q;
Contactor.Ready := (Contactor.Mode.eMode=Contactor_modes.Auto) AND True;
Contactor.Status := SEL((_w8 OR _w11) AND Inhibit_REV, SEL(_w11, _w9, eContactor_Status.Manual_Rev), eContactor_Status.REV_Limit);
_w12 := (NOT _w6 AND (_w8 OR _w11) AND Allow_Reverse) AND NOT Inhibit_REV AND NOT (Contactor.Mode.eMode=Contactor_Modes.Disabled);
Q_Rev := _w12;
Contactor.Q2 := _w12;
F_TRIG_1(CLK := TP_1.Q OR TP_0.Q); // F_trig

ACTION Status:
Contactor.Status := Sel(Inhibit_FWD, SEL(Inhibit_Rev, SEl(NOT Interlock_NC, SEL(NOT Permissive_NC, Sel((Contactor.Mode.eMode=Contactor_modes.Fwd) OR (Contactor.Mode.eMode=Contactor_modes.Bump_FWD), SEL((Contactor.Mode.eMode=Contactor_modes.Rev) OR (Contactor.Mode.eMode=Contactor_modes.Bump_REV), SEL((Contactor.Mode.eMode=Contactor_modes.Auto) AND Contactor.PLC_CMD_FWD, SEL((Contactor.Mode.eMode=Contactor_modes.Auto) AND Contactor.PLC_CMD_Rev, Contactor_Status.OFF, Contactor_Status.Auto_Rev), Contactor_Status.Auto_FWD), Contactor_Status.Manual_Rev), Contactor_Status.Manual_FWD), Contactor_Status.Interlocked), Contactor_Status.LockedOut), Contactor_Status.REV_Limit), Contactor_Status.FWD_Limit);
END_ACTION

END_FUNCTION_BLOCK

// DI_UDFB
FUNCTION_BLOCK DI_UDFB
VAR_INPUT
	Raw:BOOL;
	NC_Input:BOOL:=FALSE;
	Debounce:UINT:=500;
	EN_Alarm_State:BOOL:=TRUE;
END_VAR
VAR_OUTPUT
	//DI:Burkert.DI_DUT;
END_VAR
VAR
	TONOF_0: BURKERT_OSCAT_BASIC.TONOF;
END_VAR
VAR_IN_OUT
	//Config:LS_Config_DUT;
END_VAR
VAR_IN_OUT
	DI:Burkert.DI_DUT;
END_VAR
VAR // added by the converter: edge detectors and wires of the graphical bodies
    _w1 : TIME;
    _w2 : ANY;
    _w3 : BOOL;
END_VAR

// note: 1 stored wires end on pins the file does not list and are not shown
_w1 := UINT_TO_TIME(Debounce);
TONOF_0(IN := DI.Raw, T_ON := _w1, T_OFF := _w1); // BURKERT_OSCAT_BASIC.TONOF
_w2 := SEL(NC_INPUT AND TONOF_0.Q, SEL(NOT NC_INPUT AND NOT TONOF_0.Q, DI.Status.eStatus, DI_Status.Normal_Signal_OFF), DI_Status.Normal_Signal_Active);
DI.Raw := Raw;
_w3 := MUX(DI.Mode.eMode, TONOF_0.Q, TRUE, False);
DI.Status.eStatus := SEL(DI.MODE.eMode=DI_Modes.Forced_Off, SEL(DI.Mode.eMode=DI_Modes.Forced_On, SEL(NOT NC_Input AND TONOF_0.Q, SEL(NC_Input AND NOT TONOF_0.Q, _w2, SEL(EN_Alarm_State, Di_Status.Normal_Signal_OFF, DI_Status.Alarm_Signal_Lost)), SEL(EN_Alarm_State, Di_Status.Normal_Signal_Active, DI_Status.Alarm_Signal_Active)), DI_Status.Forced_On), DI_Status.Forced_OFF);
DI.q := _w3;

END_FUNCTION_BLOCK

// DO_UDFB
FUNCTION_BLOCK DO_UDFB
VAR_INPUT
	Lockout_NC:BOOL;
	Permisive_NC:BOOL;
	OnLine:Bool;
	
	
END_VAR
VAR_OUTPUT
	Q:BOOL;
END_VAR
VAR
END_VAR
VAR_IN_OUT
	Dout:DO_DUT;
END_VAR
VAR // added by the converter: edge detectors and wires of the graphical bodies
    _w1, _w2, _w3 : BOOL;
END_VAR

_w1 := SEL(Dout.Mode.eMode=DO_modes.Forced_On, False, True);
_w2 := Permisive_NC AND ((Dout.Mode.eMode=DO_modes.Auto) AND Dout.PLC_CMD);
_w3 := Lockout_NC AND (_w2 OR SEL(Dout.Mode.eMode=DO_modes.Forced_Off, _w1, False));
Dout.Q := _w3;
Q := _w3;
dout.Status := SEL(NOT OnLine, SEL(LockOut_NC, Do_Status.LOCKED_OUT, SEL(_w2, SEL(Dout.Mode.eMode=DO_modes.Forced_Off, SEL(_w1, SEL(permisive_NC, Do_Status.Interlocked, Do_Status.OFF), Do_Status.Forced_On), Do_Status.Forced_OFF), Do_Status.On)), Do_Status.OFFLINE);
Dout.Ready := Online AND (Dout.Mode.eMode=Do_modes.Auto);

END_FUNCTION_BLOCK

// Level_1_Devices/Burkert Library/Analog_Sensor_UDFB
FUNCTION_BLOCK Analog_Sensor_UDFB EXTENDS Analog_Alarm_UDFB
VAR_INPUT
	Alarm_Enable:BOOL:=TRUE;
	Latching:BOOL:=FALSE;
	Fault:BOOL:=FALSE;
	Online:BOOL:=TRUE;
	Raw:REAl;
END_VAR

VAR_OUTPUT
	//Status	:BYTE;
END_VAR
VAR_IN_OUT
AIT	:	Burkert.cAIT;
END_VAR

VAR
	//hihi: BOOL;
///	hi: BOOL;
	//lolo: BOOL;
	//LO: BOOL;
	//Alarm_Debounce: TON;
	//deboune_Time: TIME;
	//Alarm_Active: BOOL;
	//Alarm_Debounce_ET: TIME;
	//Alarm: BOOL;
	//ALARM_2_0: BURKERT_OSCAT_BASIC.ALARM_2;
	F_TRIG_0: F_Trig;
	TON_0: TON;
	tmpEU: REAL;
	tmpEU2: REAL;
END_VAR

VAR_TEMP
	EU_Range: REAL;
	Raw_Range: REAL;
	Corrected_Raw: REAL;
	Raw_Pct: REAL;
	EU_Scaled: REAL;
END_VAR

(* body of a kind this reader does not render *)

END_FUNCTION_BLOCK

// Level_1_Devices/Burkert Library/B8619_UDFB
FUNCTION_BLOCK B8619_UDFB
VAR_INPUT
	
END_VAR
VAR_OUTPUT
END_VAR
VAR
	Master_Scan:INT;
	Data:ARRAY[0..31] OF WORD;
	tReal:ARRAY[0..15] OF REAL;
END_VAR

METHOD PH : PH_8619
VAR_INPUT
	Raw:ARRAY[0..31] OF WORD;
END_VAR
VAR_OUTPUT
	RTD_OHM:REAL;
	Temperature:REAL;
	mv:REAL;
	ORP:REAL;
	PH_Value:REAL;
END_VAR
VAR_INST // added by the converter: edge detectors and wires of the graphical bodies
    _w1, _w2, _w3, _w4, _w5 : ANY;
END_VAR
_w1 := WORD_2_REAL_1(Low_Word := Raw[7], High_Word := Raw[6]);
RTD_OHM := _w1;
_w2 := WORD_2_REAL_1(Low_Word := Raw[9], High_Word := Raw[8]);
Temperature := _w2;
_w3 := WORD_2_REAL_1(Low_Word := Raw[11], High_Word := Raw[10]);
mv := _w3;
_w4 := WORD_2_REAL_1(Low_Word := Raw[13], High_Word := Raw[12]);
ORP := _w4;
_w5 := WORD_2_REAL_1(Low_Word := Raw[15], High_Word := Raw[14]);
PH_Value := _w5;
END_METHOD

END_FUNCTION_BLOCK

// Level_1_Devices/Burkert Library/Basic_BCV_UDFB
FUNCTION_BLOCK Basic_BCV_UDFB
VAR_INPUT
	OL:BOOL;
	CL:BOOL;
	LOCKOUT:BOOL;
	Online:BOOL;
	Interlock:BOOL;
END_VAR

VAR_OUTPUT
	Output	:BOOL;
	Output_2	:BOOL;
END_VAR

VAR_IN_OUT
	BCV	:Burkert.cBCV;
END_VAR

VAR
	Pulse:Burkert_Oscat_basic.GEN_SQ;
	TON_0:Ton;
	TOF_0:TOF;
END_VAR

Output:=Eval_Output();
Output_2:=NOT(Output);

BCV.Status:= Eval_Status();
		
		
BCV.Ready:=Eval_Ready();

METHOD Eval_Output : BOOL
VAR_INPUT
END_VAR
VAR
	
END_VAR
Pulse(PT:=T#5S);
IF Lockout THEN //OR NOT(Online) THEN
	Eval_Output:=FALSE;
ELSE
	
	CASE BCV.Mode.eMode OF
		eBCV_Modes.Open: 	Eval_Output:=TRUE;
		eBCV_Modes.Closed:	Eval_Output:=FALSE;
		eBCV_Modes.Identify: Eval_Output:=Pulse.Q;
		eBCV_Modes.Auto:
			IF Interlock THEN
				Eval_Output:=FALSE;
			ELSE
				Eval_Output:=BCV.PLC_CMD;
			END_IF;
	END_CASE;
END_IF
END_METHOD

METHOD Eval_Ready : BOOL
VAR_INPUT
	//Mode.BCV
END_VAR
Eval_Ready:=(
			BCV.Mode.eMode=eBCV_Modes.Auto AND
			Online AND
			NOT(BCV.Status=Burkert.eBCV_Status.Both_Limits_Active) AND
			NOT(BCV.Status=Burkert.eBCV_Status.Fault) AND
			NOT(BCV.Status=Burkert.eBCV_Status.Check_Function) AND
			NOT(BCV.Status=Burkert.eBCV_Status.Missing) AND
			NOT(BCV.Status=Burkert.eBCV_Status.OFFLINE) AND 
			NOT(BCV.Status=Burkert.eBCV_Status.Out_Of_Spec) AND
			NOT(BCV.Status=Burkert.eBCV_Status.P_Fault)
			);
END_METHOD

METHOD Eval_Status : eBCV_Status
VAR_INPUT

END_VAR


VAR
	lcl_Status:eBCV_Status;
END_VAR
TON_0(PT:=T#10S);
Ton_0.IN:= (
		(NOT(OL) AND NOT(CL)) OR
		(NOT(CL) AND NOT(Output)) OR
		(NOT(OL) AND Output)
		);

IF NOT(OL) AND NOT(CL) THEN
	IF Output THEN
		lcl_Status:=Burkert.eBCV_Status.Opening;
	ELSE
		lcl_Status:=Burkert.eBCV_Status.Closing;
	END_IF;
END_IF;

IF OL AND NOT(CL) THEN
	IF BCV.Mode.eMode=eBCV_Modes.Auto THEN
		lcl_Status:=Burkert.eBCV_Status.A_Open;
	ELSE
		lcl_Status:=Burkert.eBCV_Status.M_Open;
	END_IF
END_IF;

IF NOT(OL) AND CL THEN
	IF BCV.Mode.eMode=eBCV_Modes.Auto THEN
		lcl_Status:=Burkert.eBCV_Status.A_Closed;
	ELSE
		lcl_Status:=Burkert.eBCV_Status.M_Closed;
	END_IF
END_IF;

IF OL AND CL THEN
	lcl_Status:=Burkert.eBCV_Status.Both_Limits_Active;
END_IF;

IF BCV.Mode.eMode=eBCV_Modes.Auto AND Interlock THEN
	lcl_Status:=Burkert.eBCV_Status.Interlocked;
END_IF;

TOF_0(PT:=T#5S,IN:=TON_0.Q);
IF ToF_0.Q THEN
	lcl_Status:=Burkert.eBCV_Status.Fault;
END_IF;




IF NOT(Online) THEN 
	lcl_Status:= Burkert.eBCV_Status.OFFLINE; 
END_IF;
IF LOCKOUT THEN 
	lcl_Status:=Burkert.eBCV_Status.LOCKED_OUT; 
END_IF;

Eval_Status:=lcl_Status;
END_METHOD

END_FUNCTION_BLOCK

// Level_1_Devices/Burkert Library/Basic_FIT
FUNCTION_BLOCK Basic_FIT
VAR_INPUT
	//Count:DWORD;
	//Frequency:REAL;
	//Raw_Count_16Bit:BOOL;
	Rate_Units:eUnits;
	Volume_Units:eUnits;
	
	FIT:REFERENCE TO cBase_FIT;
END_VAR

VAR_OUTPUT
	Reset:BOOL;
END_VAR

VAR
	Analog_Alarm:Burkert.Analog_Alarm_UDFB;
	R_Trig_0: R_Trig;
	COUNT_REAL: LREAL;
	Total:LREAL;
	FREQUENCY_REAL: REAL;
	Rate_Sec:REAL;
	High_Word:Word;
	ALARM_1_0: BURKERT_OSCAT_BASIC.ALARM_2;
	hihi: BOOL;
	hi: BOOL;
	lolo: BOOL;
	LO: BOOL;
	Alarm_Debounce: TON;
	TON_0: TON;
END_VAR
VAR_IN_OUT
	
END_VAR

(* body of a kind this reader does not render *)

END_FUNCTION_BLOCK

// Level_1_Devices/Burkert Library/BCV_CTRL_UDFB
FUNCTION_BLOCK BCV_CTRL_UDFB
VAR_INPUT
	OL:BOOL;
	CL:BOOL;
	LOCKOUT:BOOL:=FALSE;
	Online:BOOL:=TRUE;
	Interlock:BOOL;
END_VAR

VAR_OUTPUT
	Output	:BOOL;
	Output_2	:BOOL;
END_VAR

VAR_IN_OUT
	BCV	:Burkert.cBCV;
END_VAR

VAR  
	Pulse_0: Burkert_OSCAT_BASIC.GEN_SQ;
	
END_VAR

(* body of a kind this reader does not render *)

END_FUNCTION_BLOCK

// Level_1_Devices/Burkert Library/FIT_Count_UDFB
FUNCTION_BLOCK FIT_Count_UDFB
VAR_INPUT
	Count:DWORD;
	//K:REAL;
	Raw_Count_16Bit:BOOL:=TRUE;
	Rate_Units:eUnits;
	Volume_Units:eUnits;
END_VAR

VAR_OUTPUT
	Reset:BOOL;
END_VAR

VAR
	R_Trig_0: R_Trig;
	COUNT_REAL: LREAL;
	Total:LREAL;
	FREQUENCY_REAL: REAL;
	Rate_Sec:REAL;
	High_Word:Word;
	ALARM_1_0: BURKERT_OSCAT_BASIC.ALARM_2;
	hihi: BOOL;
	hi: BOOL;
	lolo: BOOL;
	LO: BOOL;
	Alarm_Debounce: TON;
	//TON_0: TON;
	Pulse_500ms:Burkert_OSCAT_BASIC.CLK_PRG;
	Pulse_1s:Burkert_OSCAT_BASIC.CLK_PRG;
	tCount:DWORD;
	Analog_Alarm:Burkert.Analog_Alarm_UDFB;
	Reset_Ton:TON;
	Count_Change:ARRAY[0..4] OF INT;
	Count_Index:INT;
	Ave_Hz:REAL;
	Calculate_Hz: CalculateFrequencyWithTime;
	Hz_1: REAL;
	Hz2: REAL;
	Count_2_Hz: Count_to_hz;
END_VAR
VAR_IN_OUT
	FIT:Burkert.cFIT;
END_VAR

(* body of a kind this reader does not render *)

END_FUNCTION_BLOCK

// Level_1_Devices/Burkert Library/FIT_Rate_UDFB
FUNCTION_BLOCK FIT_Rate_UDFB
VAR_INPUT
	//Count:DWORD;
	Frequency:REAL;
	Rate_Units:eUnits;
	Volume_Units:eUnits;
END_VAR

VAR_OUTPUT
	//Reset:BOOL;
END_VAR

VAR
	Analog_Alarm:Burkert.Analog_Alarm_UDFB;
	R_Trig_0: R_Trig;
	COUNT_REAL: LREAL;
	Total:LREAL;
	FREQUENCY_REAL: REAL;
	Rate_Sec:REAL;
	High_Word:Word;
	ALARM_1_0: BURKERT_OSCAT_BASIC.ALARM_2;
	hihi: BOOL;
	hi: BOOL;
	lolo: BOOL;
	LO: BOOL;
	Alarm_Debounce: TON;
	TON_0: TON;
	Pulse_1s:Burkert_OSCAT_BASIC.CLK_PRG;
	tCount:REAL;
	
END_VAR
VAR_IN_OUT
	FIT:Burkert.cFIT;
	
	
END_VAR

(* body of a kind this reader does not render *)

END_FUNCTION_BLOCK

// Level_1_Devices/Burkert Library/FIT_UDFB
FUNCTION_BLOCK FIT_UDFB
VAR_INPUT
	Count:DWORD;
	Frequency:REAL;
	Raw_Count_16Bit:BOOL;
	Rate_Units:eUnits;
	Volume_Units:eUnits;
END_VAR

VAR_OUTPUT
	Reset:BOOL;
END_VAR

VAR
	Analog_Alarm:Burkert.Analog_Alarm_UDFB;
	R_Trig_0: R_Trig;
	COUNT_REAL: LREAL;
	Total:LREAL;
	FREQUENCY_REAL: REAL;
	Rate_Sec:REAL;
	High_Word:Word;
	ALARM_1_0: BURKERT_OSCAT_BASIC.ALARM_2;
	hihi: BOOL;
	hi: BOOL;
	lolo: BOOL;
	LO: BOOL;
	Alarm_Debounce: TON;
	TON_0: TON;
END_VAR
VAR_IN_OUT
	FIT:Burkert.cFIT;
END_VAR

(* body of a kind this reader does not render *)

END_FUNCTION_BLOCK

// Level_1_Devices/Burkert Library/LS_UDFB
FUNCTION_BLOCK LS_UDFB
VAR_INPUT
	Wired_NC:BOOL;
	On_Delay_ms:UINT;
	Off_Delay_ms:UINT;
	Alarm_Dry:BOOL;
	Alarm_Wet:BOOL;
	Raw:BOOL;
	Device: REFERENCE TO Burkert.DI_DUT;
END_VAR
VAR_OUTPUT
END_VAR
	

VAR
	TON_0:TON;
	TOF_0:TOF;
	LCL_raw:Bool;
END_VAR

VAR_IN_OUT
	//Device:Burkert.DI_DUT;
END_VAR

Device.Raw:=Raw;
CASE Device.MODE.eMode OF 
	DI_Modes.Auto: 			LCL_Raw:=Device.Raw;
	DI_Modes.Forced_Off:	LCL_Raw:=FALSE;
	DI_Modes.Forced_On:		LCL_Raw:=TRUE;
END_CASE

TON_0(PT:=(TO_TIME(On_Delay_ms)),IN:=LCL_RAW);
TOF_0(PT:=(TO_TIME(Off_Delay_ms)),IN:=TON_0.Q,Q=>Device.Q);


IF Wired_NC THEN
	Device.Status.eStatus:=SEL(Device.Q,DI_Status.Liquid_Detected,DI_Status.No_Liquid_Detected);
ELSE
	Device.Status.eStatus:=SEL(Device.Q,DI_Status.NO_Liquid_Detected,DI_Status.Liquid_Detected);
END_IF;

IF Alarm_Dry AND Device.Status.eStatus=DI_Status.NO_Liquid_Detected THEN
	Device.Status.eStatus:=DI_Status.No_Liquid_Detected_Alarm;
END_IF;

IF Alarm_Wet AND Device.Status.eStatus=DI_Status.Liquid_Detected THEN
	Device.Status.eStatus:=DI_Status.Liquid_Detected_Alarm;
END_IF;

END_FUNCTION_BLOCK

// Level_1_Devices/Burkert Library/SV_Fun
FUNCTION SV_Fun :BOOL;
VAR_INPUT
	Lockout_NC:BOOL;
	Permisive_NC:BOOL;
	Online:BOOL;
	Normally_Open_Valve:BOOL:=FALSE;;
	
	
END_VAR
VAR_OUTPUT
	//Q:BOOL;
END_VAR
VAR
END_VAR
VAR_IN_OUT
	SV:SV_DUT;
END_VAR
VAR // added by the converter: edge detectors and wires of the graphical bodies
    _w1, _w2, _w3, _w5, _w6 : BOOL;
    _w4 : ANY;
END_VAR

_w1 := SEL(SV.Mode.eMode=eBCV_Modes.Open, False, True);
_w2 := Permisive_NC AND ((SV.Mode.eMode=eBCV_Modes.Auto) AND SV.PLC_CMD);
_w3 := _w2 OR SEL(SV.Mode.eMode=eBCV_Modes.Closed, _w1, False);
_w4 := Burkert_OSCAT_BASIC.REPLACE_ALL(str := TO_String(SV.Namur.eNamur), src := '_', rep := ' ');
SV.strNamur := _w4;
_w5 := Lockout_NC AND _w3;
_w6 := SEL(Normally_Open_Valve, _w5, NOT _w5);
SV.Q := _w6;
SV_Fun := _w6;
SV.Status := SEL(NOT Online, SEL(LockOut_NC, Burkert.eBCV_Status.LOCKED_OUT, SEL(_w2, SEL(SV.Mode.eMode=eBCV_Modes.Closed, SEL(_w1, SEL(permisive_NC, Burkert.eBCV_Status.Interlocked, Burkert.eBCV_Status.A_Closed), Burkert.eBCV_Status.M_Open), Burkert.eBCV_Status.M_Closed), Burkert.eBCV_Status.A_Open)), Burkert.eBCV_Status.OFFLINE);
SV.Ready := (SV.Mode.eMode=eBCV_Modes.Auto) AND True AND Online;
// LockOut_NC: input not connected

END_FUNCTION

// Analog_Pump
FUNCTION_BLOCK Analog_Pump
VAR_INPUT
	Device:REFERENCE TO cAnalog_Pump;
	Lockout_NC:BOOL;
	Permissive_NC:BOOL;
END_VAR
VAR_OUTPUT
	FWD:BOOL;
	REV:BOOL;
	CV:REAL;
END_VAR
VAR
END_VAR



CASE Device.Mode.eMode OF
	
	eAnalog_Pump_Modes.Disabled:
		FWD:=FALSE;
		REV:=FALSE;
		CV:=0;
	eAnalog_Pump_Modes.Manual:
		CV:=Device.HMI_Rate_PCT;
		IF CV>1 THEN
			FWD:=TRUE;
			REV:=FALSE;
		END_IF
		IF CV < (-1) THEN
			FWD:=FALSE;
			REV:=TRUE;
		END_IF
	eAnalog_Pump_Modes.Auto:
		IF Device.PLC_Run THEN
			CV:=Device.PLC_Rate_PCT;
			FWD:=Device.PLC_Run;
			Rev:=FALSE;
		ELSE
			FWD:=FALSE;
			REV:=FALSE;
			CV:=0;
		END_IF;
			
		
END_CASE

IF NOT(lockout_NC)  OR ( NOT(Permissive_NC) AND Device.Mode.eMode=eAnalog_Pump_Modes.Auto) OR NOT(Device.Healthy)  THEN
	FWD:=FALSE;
	REV:=FALSE;
	CV:=0;
END_IF

Device.Pump_CV:=CV;
Device.PUMP_FWD:=FWD;
Device.PUMP_REV:=REV;

Status();

ACTION Status:
Device.Status.eStatus:=eAnalog_Pump_Status.IDLE	;

IF device.Mode.eMode=eAnalog_Pump_Modes.Disabled THEN		device.Status.eStatus:=	eAnalog_pump_Status.Disabled; 	END_IF;
IF Device.Mode.eMode=eAnalog_Pump_Modes.Manual THEN			Device.Status.eStatus:=eAnalog_pump_Status.Manual;		END_IF;



IF Device.Actual>1 AND Device.Pump_CV>1 THEN
	IF Device.Mode.eMode=eAnalog_Pump_Modes.Auto THEN Device.Status.eStatus:=eAnalog_pump_Status.Running; END_IF;
	IF Device.Mode.eMode=eAnalog_Pump_Modes.Manual THEN Device.Status.eStatus:=eAnalog_pump_Status.Manual; END_IF;
END_IF

IF NOT(Permissive_NC) AND Device.Mode.eMode=eAnalog_Pump_Modes.Auto THEN Device.Status.eStatus:=eAnalog_pump_Status.Interlocked; END_IF;



IF Device.Mode.eMode=eAnalog_Pump_Modes.Prime THEN			Device.Status.eStatus:=eAnalog_pump_Status.Prime;		END_IF;




IF NOT(Lockout_NC) THEN
	Device.Status.eStatus:=eAnalog_Pump_Status.Locked_Out;
END_IF;

IF NOT(Device.Healthy) THEN
	Device.Status.eStatus:=eAnalog_Pump_Status.Fault;
END_IF;
IF Device.Actual<(-1) THEN Device.Status.eStatus:=eAnalog_Pump_Status.Fault; END_IF;
IF Device.Actual>(101) THEN Device.Status.eStatus:=eAnalog_Pump_Status.Fault; END_IF;

Device.Actual:= SEL(FPU.IsRealNaN(Device.Actual ),Device.Actual,-999);
Device.Ready:=Device.Mode.eMode=eAnalog_Pump_Modes.Auto AND Device.Healthy AND Device.Actual>(-1) AND Device.Actual<(101);
END_ACTION

END_FUNCTION_BLOCK

// Eaton_DM1
FUNCTION_BLOCK Eaton_DM1
VAR_INPUT
	Interlock_NC:BOOL;
	Permissive_NC:BOOL;
	CommState:ModbusTCPComState;
	VFD: REFERENCE TO cVFD_Eaton_DUT;
	Current_Alarm_EN:BOOL:=FALSE;
END_VAR
VAR_OUTPUT
END_VAR
VAR
	VFD_Run:BOOL;
	VFD_CMD_PCT:REAL;
	//T_1m: Burkert_OSCAT_BASIC.CLK_PRG;
	lclAlarm_Active:RS;
	Alarm:Burkert.Analog_Alarm_UDFB;
	lclStatus:eVFD_Status;
END_VAR




Data_In();
Control();
Status();
Data_Out();


//T_1m(PT:=T#60s);

ACTION Control:
CASE VFD.MODE.eMode OF 
	eVFD_Modes.Auto:
		VFD.MAN_CMD:=VFD.PLC_CMD;
		IF Permissive_NC THEN	
			VFD_CMD_PCT:=VFD.PLC_CMD;
			VFD_Run:=VFD.PLC_Run;
		ELSE
			VFD_CMD_PCT:=0;
			VFD_Run:=FALSE;
		END_IF;
	eVFD_Modes.Disabled:
		VFD_CMD_PCT:=0;
		VFD_Run:=FALSE;
	eVFD_Modes.Manual:
		VFD_CMD_PCT:=VFD.MAN_CMD;
		VFD_Run:=(VFD.MAN_CMD<(-10) OR VFD.MAN_CMD>10);
	eVFD_Modes.Reset:
		VFD_CMD_PCT:=0;
		VFD_Run:=FALSE;
		
	eVFD_Modes.Simulate:
		VFD.MAN_CMD:=VFD.PLC_CMD;
		IF Permissive_NC THEN	
			VFD_CMD_PCT:=VFD.PLC_CMD;
			VFD_Run:=VFD.PLC_Run;
		ELSE
			VFD_CMD_PCT:=0;
			VFD_Run:=FALSE;
		END_IF;
END_CASE;

IF NOT(Interlock_NC) THEN
	VFD_CMD_PCT:=0;
	VFD_Run:=FALSE;
END_IF;
END_ACTION

ACTION Data_IN:
//Status_Word RX[0]
VFD.Data.Drive_STATUS.Ready:=VFD.RX[0].0;
VFD.Data.Drive_STATUS.Run:=VFD.RX[0].1;
VFD.Data.Drive_STATUS.FWD:=NOT(VFD.RX[0].2);
VFD.Data.Drive_STATUS.Fault:=VFD.RX[0].3;
VFD.Data.Drive_STATUS.alarm:=VFD.RX[0].4;
VFD.Data.Drive_STATUS.At_Speed:=VFD.RX[0].5;


//General Status RX[1]
VFD.Data.Drive_STATUS.FieldBus:=VFD.RX[1].12;
VFD.Data.Drive_STATUS.Flux_Ready:=VFD.RX[1].7;


//Actual Speed RX[2]
VFD.Output_Pct:=TO_REAL(VFD.RX[2])/100; 


VFD.Output_Hz:=TO_REAL(VFD.RX[3])/1000;
VFD.Data.RPM:=TO_INT(VFD.RX[4]);
VFD.Data.Motor_Current:=TO_REAL(VFD.RX[5])/1000;
VFD.Data.Motor_Torque:=TO_REAL(TO_INT(VFD.RX[6]))/10;
VFD.Data.Motor_Power:=TO_REAL(VFD.RX[7])/10;
VFD.Data.Motor_Voltage:=TO_REAL(VFD.RX[8])/10;
VFD.Data.DC_Link:=TO_REAL(VFD.RX[9]);
VFD.Data.Fault_Code:=TO_INT(VFD.RX[10]);
	
//VFD.a
VFD.Control.Actual:=VFD.Output_Pct;

IF VFD.Control.MODE.eMode=eVFD_Modes.Simulate THEN 
	VFD.Data.Drive_STATUS.Fault:=FALSE;
	VFD.Data.Drive_STATUS.At_Speed:=(VFD.Output_Hz>5);
	
	VFD.RX[0].0:=TRUE;	//VFD.Data.Drive_STATUS.Ready:=
	VFD.RX[0].1:=VFD.TX[0].0;		//VFD.Data.Drive_STATUS.Run:=
	VFD.RX[0].2:=VFD.TX[0].1;	//VFD.Data.Drive_STATUS.FWD:=
	
	IF VFD.TX[0].0 THEN
		VFD.RX[2]:=VFD.TX[2];	//VFD.Control.Output_Pct:=
		VFD.RX[3]:=TO_WORD(TO_REAL(VFD.TX[2]/1.66));		//VFD.Control.Output_Hz:=TO_REAL(
	ELSE
		VFD.RX[2]:=0;
		VFD.RX[3]:=0;
	END_IF;
	
	VFD.RX[9]:=624;	//VFD.Data.DC_Link:=TO_REAL(
	
END_IF;
END_ACTION

ACTION Data_Out:
//TX[0]- FB Control Word







VFD.TX[0]:=0;
VFD.TX[0].0:=VFD_Run;
VFD.TX[0].1:=(VFD_CMD_PCT<0) ;//AND Allow_Reverse;

VFD.TX[0].2:=VFD.MODE.eMode=eVFD_Modes.Reset;
VFD.TX[0].3:=FALSE;
VFD.TX[0].4:=FALSE;
VFD.TX[0].5:=FALSE;
VFD.TX[0].6:=FALSE;
VFD.TX[0].7:=FALSE;
//VFD.TX[0].8:=TRUE;//NOT(VFD.MODE.eMode=eVFD_Modes.Disabled); //FB Control On
//VFD.TX[0].9:=TRUE;//NOT(VFD.MODE.eMode=eVFD_Modes.Disabled);	//FB Reference ON


//TX[1] FB General Control Word; Not USed
VFD.TX[1]:=0;
//TX[2] Speed Reference
VFD.TX[2]:=TO_WORD(ABS((VFD_CMD_PCT)*100));
END_ACTION

ACTION Status:
lclAlarm_Active(Reset1:=(VFD.MODE.eMode=eVFD_Modes.Reset OR NOT(Current_Alarm_EN) ));

VFD.Ready:=(
	(CommState=ModbusTCPComState.CONNECTED OR CommState=ModbusTCPComState.OFF) AND 
	(VFD.MODE.eMode=eVFD_Modes.Auto OR VFD.MODE.eMode=eVFD_Modes.Simulate) AND 
	VFD.Data.Drive_STATUS.Ready AND
	NOT(lclAlarm_Active.Q1) );
	
VFD.Status.eStatus:=eVFD_Status.READY;



IF VFD.Data.Drive_STATUS.Run AND VFD.MODE.eMode=eVFD_Modes.Manual AND VFD.Data.Drive_STATUS.At_Speed THEN	VFD.Status.eStatus:=eVFD_Status.M_Runing; END_IF;
IF VFD.Data.Drive_STATUS.Run AND VFD.MODE.eMode=eVFD_Modes.Auto AND VFD.Data.Drive_STATUS.At_Speed THEN VFD.Status.eStatus:=eVFD_Status.A_Running; END_IF;
IF VFD.Data.Drive_STATUS.Run AND VFD.MODE.eMode=eVFD_Modes.Simulate AND VFD.Data.Drive_STATUS.At_Speed THEN VFD.Status.eStatus:=eVFD_Status.A_Running; END_IF;
IF VFD.Data.Drive_STATUS.Run  AND NOT(VFD.Data.Drive_STATUS.At_Speed) THEN VFD.Status.eStatus:=eVFD_Status.Ramping; END_IF;
IF VFD.MODE.eMode=eVFD_Modes.Auto AND NOT(Permissive_NC) THEN VFD.Status.eStatus:=eVFD_Status.Interlocked; END_IF;

IF VFD.Data.Drive_STATUS.Fault THEN 
	VFD.Status.eStatus:=eVFD_Status.Fault; 
	VFD_CMD_PCT:=0;
	VFD_Run:=FALSE;
END_IF;

IF VFD.MODE.eMode=eVFD_Modes.Disabled THEN VFD.Status.eStatus:=eVFD_Status.Disabled; END_IF;
IF NOT(Permissive_NC) THEN 	VFD.Status.eStatus:=eVFD_Status.Interlocked; END_IF;
IF NOT(Interlock_NC) THEN 
		VFD.Status.eStatus:=eVFD_Status.LOCKED_OUT; 
		VFD_CMD_PCT:=0;
		VFD_Run:=FALSE;
END_IF;



IF VFD.Data.DC_Link<100 THEN	VFD.Status.eStatus:=eVFD_Status.Low_Voltage; END_IF;
IF VFD.Data.Fault_Code=66 THEN VFD.Status.eStatus:=eVFD_Status.Safe_Torque_Off; END_IF;

IF NOT(CommState=ModbusTCPComState.CONNECTED OR CommState=ModbusTCPComState.OFF)	AND NOT(VFD.MODE.eMode=eVFD_Modes.Simulate)	THEN 
	VFD.Status.eStatus:=eVFD_Status.Offline;
	VFD_CMD_PCT:=0;
	VFD.Output_Pct:=0;
	VFD_Run:=FALSE;
END_IF;


CASE CommState OF
	ModbusTCPComState.OFF: 			VFD.strTCPstate:='OFF';
	ModbusTCPComState.CONNECTING: 	VFD.strTCPstate:='CONNECTING';
	ModbusTCPComState.CONNECTED: 	VFD.strTCPstate:='CONNECTED';
	ModbusTCPComState.DISCONNECTING: VFD.strTCPstate:='DISCONNECTING';
	ModbusTCPComState.SOCKET_ERROR: VFD.strTCPstate:='SOCKET_ERROR';
END_CASE



VFD.Current_Alarm.Silence:=VFD.Output_Pct<25;
Alarm(Config:=VFD.Current_Alarm,eu:=VFD.Data.Motor_Current,Debounce_Active:=FALSE,status=>VFD.Current_Status.eStatus);
lclAlarm_Active.SET:=FALSE;
IF Current_Alarm_EN THEN
	CASE Alarm.Status OF
		Burkert.eSensor_Status.HiHi_Alarm:
			VFD.Status.eStatus:=eVFD_Status.High_High_Current_Alarm;
			lclStatus:=VFD.Status.eStatus;
			lclAlarm_Active.SET:=TRUE;
		Burkert.eSensor_Status.High_Warning:
			VFD.Status.eStatus:=eVFD_Status.High_Current_Warning;
			//lclStatus:=VFD.Status.eStatus;
			//lclAlarm_Active.SET:=TRUE;
		Burkert.eSensor_Status.Low_Warning:
			VFD.Status.eStatus:=eVFD_Status.Low_Current_Warning;
			//lclStatus:=VFD.Status.eStatus;
			//lclAlarm_Active.SET:=TRUE;
		Burkert.eSensor_Status.Low_Low_Alarm:
			VFD.Status.eStatus:=eVFD_Status.Low_Low_Current_Alarm;
			lclStatus:=VFD.Status.eStatus;
			lclAlarm_Active.SET:=TRUE;
	END_CASE
END_IF;

IF VFD.Output_Pct>50 AND VFD.Data.Motor_Current<0.1 THEN
	VFD.Status.eStatus:=eVFD_Status.No_Motor_Load_Detected;
	lclStatus:=VFD.Status.eStatus;
	lclAlarm_Active.SET:=TRUE;
END_IF;

IF lclAlarm_Active.Q1 THEN
	VFD.Status.eStatus:=lclStatus;
	VFD_CMD_PCT:=0;
	VFD_Run:=FALSE;
END_IF;

(*
T_1m(PT:=T#60S);
IF T_1m.Q AND VFD.Data.Drive_STATUS.Run THEN
	VFD.RunTime_Minutes:=VFD.RunTime_Minutes+1;
END_IF;
*)
END_ACTION

END_FUNCTION_BLOCK

// Nord_VFD_UDFB
FUNCTION_BLOCK Nord_VFD_UDFB
VAR_INPUT
	Interlock:BOOL;
	Permissive:BOOL;
	//Online:BOOL;
	Allow_Reverse:Bool;
END_VAR
VAR_OUTPUT
END_VAR
VAR
END_VAR
VAR_IN_OUT
	Nord_VFD:cNord_VFD;
END_VAR
VAR // added by the converter: edge detectors and wires of the graphical bodies
    _w1, _w2, _w3 : ANY;
    _w4, _w5 : BOOL;
END_VAR

fNord_Status_Mapping(Raw := Nord_VFD.Status.Status_Word.RAW, Status => _w1);
Nord_VFD.Status.Status_Word := _w1;
_w2 := fNord_Control_Word(Control := Nord_VFD.Control);
Nord_VFD.Control.Raw := _w2;
_w3 := BURKERT_OSCAT_BASIC.SCALE_R(X := UINT_TO_REAL(Nord_VFD.Status.Actual_Frequency), I_LO := -16384, I_HI := 16384, O_LO := (-100.0), O_HI := 100.0);
Nord_VFD.Ouput_PCT := _w3;
_w4 := Interlock AND True AND (Nord_VFD.Mode=eVFD_Modes.Manual);
_w5 := (Nord_VFD.Mode=eVFD_Modes.Auto) AND Interlock AND Permissive AND TRUE AND Nord_VFD.PLC_Run;
Nord_VFD.Control.Ready_For_Operation := _w5 OR _w4;
Nord_VFD.SP_TX := REAL_TO_INT(SEL(_w4, SEL(_w5, 0.0, Nord_VFD.PLC_SP), Nord_VFD.MAN_SP) * 163.84);
Nord_VFD.Control.Emergency_Stop := TRUE;
Nord_VFD.Control.Enable_pulses := TRUE;
Nord_VFD.Control.Enable_Ramp := TRUE;
Nord_VFD.Control.Enable_Setpoint := TRUE;
Nord_VFD.Control.Enable_Voltage := TRUE;
Nord_VFD.Control.Control_Data_Valid := TRUE;
Nord_VFD.Control.Enable_Operation := TRUE;
Nord_VFD.Control.ACK_Error := Nord_VFD.Mode=eVFD_Modes.Reset;
Nord_VFD.eStatus := SEL(Nord_VFD.Status.Status_Word.Fault, SEL(Nord_VFD.Status.Status_Word.Enabled AND Nord_VFD.Status.Status_Word.Setpoint_Reached, SEL(Nord_VFD.Status.Status_Word.Enabled AND NOT Nord_VFD.Status.Status_Word.Setpoint_Reached, SEL(Nord_VFD.Status.Status_Word.Ready_to_Start, eVFD_Status.Offline, eVFD_Status.READY), eVFD_Status.Ramping), eVFD_Status.A_Running), eVFD_Status.Fault);

END_FUNCTION_BLOCK

// Vacon_100
FUNCTION_BLOCK Vacon_100
VAR_INPUT
	Interlock_NC:BOOL;
	Permissive_NC:BOOL;
	Allow_Reverse:BOOL:=FALSE;
	Max_Hz:REAL:=60;
	CommState:ModbusTCPComState;
	Current_Alarm_EN:BOOL:=FALSE;
END_VAR
VAR_OUTPUT
END_VAR
VAR_IN_OUT
	VFD	:	cVFD_Vacon;
END_VAR


VAR
	VFD_Run:BOOL;
	VFD_CMD_PCT:REAL;
	T_1m: Burkert_OSCAT_BASIC.CLK_PRG;
	lclAlarm_Active:RS;
	Alarm:Burkert.Analog_Alarm_UDFB;
	lclStatus:eVFD_Status;
END_VAR




Data_In();
Control();
Status();
Data_Out();


T_1m(PT:=T#60s);

ACTION Control:
CASE VFD.Control.MODE.eMode OF 
	eVFD_Modes.Auto:
		VFD.Control.MAN_CMD:=VFD.Control.PLC_CMD;
		IF Permissive_NC THEN	
			VFD_CMD_PCT:=VFD.Control.PLC_CMD;
			VFD_Run:=VFD.Control.PLC_Run;
		ELSE
			VFD_CMD_PCT:=0;
			VFD_Run:=FALSE;
		END_IF;
	eVFD_Modes.Disabled:
		VFD_CMD_PCT:=0;
		VFD_Run:=FALSE;
	eVFD_Modes.Manual:
		VFD_CMD_PCT:=VFD.Control.MAN_CMD;
		VFD_Run:=(VFD.Control.MAN_CMD<(-10) OR VFD.Control.MAN_CMD>10);
	eVFD_Modes.Reset:
		VFD_CMD_PCT:=0;
		VFD_Run:=FALSE;
		
	eVFD_Modes.Simulate:
		VFD.Control.MAN_CMD:=VFD.Control.PLC_CMD;
		IF Permissive_NC THEN	
			VFD_CMD_PCT:=VFD.Control.PLC_CMD;
			VFD_Run:=VFD.Control.PLC_Run;
		ELSE
			VFD_CMD_PCT:=0;
			VFD_Run:=FALSE;
		END_IF;
END_CASE;

IF NOT(Interlock_NC) THEN
	VFD_CMD_PCT:=0;
	VFD_Run:=FALSE;
END_IF;
END_ACTION

ACTION Data_IN:
VFD.Data.Status_code:=VFD.rx[0];


VFD.Data.Drive_STATUS.Ready:=	VFD.rx[0].0;
VFD.Data.Drive_STATUS.Run:=		VFD.rx[0].1;
VFD.Data.Drive_Status.FWD:=		VFD.rx[0].2;
VFD.Data.Drive_Status.Fault:=	VFD.rx[0].3;
VFD.Data.Drive_Status.Alarm:=	VFD.rx[0].4;
VFD.Data.Drive_Status.At_Speed:=	VFD.rx[0].5;
VFD.Data.Drive_Status.Zero_Speed:=	VFD.rx[6].6;
VFD.Data.Drive_Status.Flux_Ready:=	VFD.rx[0].7;

VFD.Data.Drive_STATUS.FieldBus	:= NOT(VFD.rx[1].13) AND NOT(VFD.rx[1].14) AND VFD.rx[1].15;
VFD.Data.Drive_Status.Keypad	:=	NOT(VFD.rx[1].13) AND (VFD.rx[1].14) AND NOT(VFD.rx[1].15);
VFD.Data.Drive_Status.PC		:=	NOT(VFD.rx[1].13) AND (VFD.rx[1].14) AND (VFD.rx[1].15);
VFD.Data.Drive_Status.Terminals	:=	NOT(VFD.rx[1].13) AND NOT(VFD.rx[1].14) AND NOT(VFD.rx[1].15);


VFD.Data.RPM:=VFD.rx[4];
Data.tWord:=VFD.RX[3];
VFD.Output_Hz:=TO_REAL(Data.tInt)/100;
VFD.Data.Motor_Current:=Word_2_real_DIV(WD:=VFD.RX[5],rDiv:=100);
VFD.Data.Motor_Torque:=Word_2_real_DIV(WD:=VFD.RX[6],rDiv:=10);
VFD.Data.Unit_Temperature:=Word_2_real_DIV(WD:=VFD.RX[7],rDiv:=10);
VFD.Data.Motor_Voltage:=Word_2_real_DIV(WD:=VFD.RX[8],rDiv:=10);

VFD.Data.DC_Link:=VFD.rx[9];
VFD.Data.Fault_Code:=VFD.rx[10];

VFD.Control.Actual:=VFD.Output_Pct;

IF VFD.Control.MODE.eMode=eVFD_Modes.Simulate THEN 
	VFD.Data.Drive_STATUS.Fault:=FALSE;
	VFD.Data.Drive_STATUS.At_Speed:=(vfd.Output_Hz>5);
	
	VFD.RX[0].0:=TRUE;	//VFD.Data.Drive_STATUS.Ready:=
	VFD.RX[0].1:=VFD.TX[0].0;		//VFD.Data.Drive_STATUS.Run:=
	VFD.RX[0].2:=VFD.TX[0].1;	//VFD.Data.Drive_STATUS.FWD:=
	
	IF VFD.TX[0].0 THEN
		VFD.RX[2]:=VFD.TX[2];	//VFD.Output_Pct:=
		VFD.RX[3]:=TO_WORD(TO_REAL(VFD.TX[2]/1.66));		//vfd.Output_Hz:=TO_REAL(
	ELSE
		VFD.RX[2]:=0;
		VFD.RX[3]:=0;
	END_IF;
	
	VFD.RX[9]:=624;	//VFD.Data.DC_Link:=TO_REAL(
	
END_IF;
END_ACTION

ACTION Data_Out:
//TX[0]- FB Control Word
VFD.TX[0]:=0;
VFD.TX[0].0:=VFD_Run;
VFD.TX[0].1:=(VFD_CMD_PCT<0) AND Allow_Reverse;
VFD.TX[0].2:=VFD.Control.MODE.eMode=eVFD_Modes.Reset;
VFD.TX[0].3:=FALSE;
VFD.TX[0].4:=FALSE;
VFD.TX[0].5:=FALSE;
VFD.TX[0].6:=FALSE;
VFD.TX[0].7:=FALSE;
VFD.TX[0].8:=TRUE;//NOT(VFD.MODE.eMode=eVFD_Modes.Disabled); //FB Control On
VFD.TX[0].9:=TRUE;//NOT(VFD.MODE.eMode=eVFD_Modes.Disabled);	//FB Reference ON


//TX[1] FB General Control Word; Not USed
VFD.TX[1]:=0;
//TX[2] Speed Reference
VFD.TX[2]:=TO_WORD(ABS((VFD_CMD_PCT)*100));
END_ACTION

ACTION Data_Sim:



IF Permissive_NC THEN	
	VFD_CMD_PCT:=VFD.Control.PLC_CMD;
	VFD_Run:=VFD.Control.PLC_Run;
ELSE
	VFD_CMD_PCT:=0;
	VFD_Run:=FALSE;
END_IF;

VFD.Output_Hz:= VFD_CMD_PCT *(Max_Hz/100);
VFD.Data.Drive_STATUS.Ready:=TRUE;
VFD.Data.Drive_STATUS.Fault:=FALSE;
VFD.Data.DC_Link:=110;
VFD.Data.Fault_Code:=000;
VFD.CONTROL.Actual:=VFD_CMD_PCT;

CommState:=ModbusTCPComState.CONNECTED;
END_ACTION

ACTION Status:
lclAlarm_Active(Reset1:=(VFD.Control.MODE.eMode=eVFD_Modes.Reset OR NOT(Current_Alarm_EN) ));

VFD.Control.Ready:=(
	(CommState=ModbusTCPComState.CONNECTED OR CommState=ModbusTCPComState.OFF) AND 
	(VFD.Control.MODE.eMode=eVFD_Modes.Auto OR VFD.Control.MODE.eMode=eVFD_Modes.Simulate) AND 
	VFD.Data.Drive_STATUS.Ready AND
	NOT(lclAlarm_Active.Q1) );
	
VFD.Status.eStatus:=eVFD_Status.READY;



IF VFD.Data.Drive_STATUS.Run AND VFD.Control.MODE.eMode=eVFD_Modes.Manual AND VFD.Data.Drive_STATUS.At_Speed THEN	VFD.Status.eStatus:=eVFD_Status.M_Runing; END_IF;
IF VFD.Data.Drive_STATUS.Run AND VFD.Control.MODE.eMode=eVFD_Modes.Auto AND VFD.Data.Drive_STATUS.At_Speed THEN VFD.Status.eStatus:=eVFD_Status.A_Running; END_IF;
IF VFD.Data.Drive_STATUS.Run AND VFD.Control.MODE.eMode=eVFD_Modes.Simulate AND VFD.Data.Drive_STATUS.At_Speed THEN VFD.Status.eStatus:=eVFD_Status.A_Running; END_IF;
IF VFD.Data.Drive_STATUS.Run  AND NOT(VFD.Data.Drive_STATUS.At_Speed) THEN VFD.Status.eStatus:=eVFD_Status.Ramping; END_IF;
IF VFD.Control.MODE.eMode=eVFD_Modes.Auto AND NOT(Permissive_NC) THEN VFD.Status.eStatus:=eVFD_Status.Interlocked; END_IF;

IF VFD.Data.Drive_STATUS.Fault THEN 
	VFD.Status.eStatus:=eVFD_Status.Fault; 
	VFD_CMD_PCT:=0;
	VFD_Run:=FALSE;
END_IF;

IF VFD.Control.MODE.eMode=eVFD_Modes.Disabled THEN VFD.Status.eStatus:=eVFD_Status.Disabled; END_IF;
IF NOT(Permissive_NC) THEN 	VFD.Status.eStatus:=eVFD_Status.Interlocked; END_IF;
IF NOT(Interlock_NC) THEN 
		VFD.Status.eStatus:=eVFD_Status.LOCKED_OUT; 
		VFD_CMD_PCT:=0;
		VFD_Run:=FALSE;
END_IF;



IF VFD.Data.DC_Link<100 THEN	VFD.Status.eStatus:=eVFD_Status.Low_Voltage; END_IF;
IF VFD.Data.Fault_Code=66 THEN VFD.Status.eStatus:=eVFD_Status.Safe_Torque_Off; END_IF;

IF NOT(CommState=ModbusTCPComState.CONNECTED OR CommState=ModbusTCPComState.OFF)	AND NOT(VFD.Control.MODE.eMode=eVFD_Modes.Simulate)	THEN 
	VFD.Status.eStatus:=eVFD_Status.Offline;
	VFD_CMD_PCT:=0;
	VFD.Output_Pct:=0;
	VFD_Run:=FALSE;
END_IF;


CASE CommState OF
	ModbusTCPComState.OFF: VFD.strTCPstate:='OFF';
	ModbusTCPComState.CONNECTING: VFD.strTCPstate:='CONNECTING';
	ModbusTCPComState.CONNECTED: VFD.strTCPstate:='CONNECTED';
	ModbusTCPComState.DISCONNECTING: VFD.strTCPstate:='DISCONNECTING';
	ModbusTCPComState.SOCKET_ERROR: VFD.strTCPstate:='SOCKET_ERROR';
END_CASE



VFD.Control.Current_Alarm.Silence:=VFD.Output_Pct<25;
Alarm(Config:=VFD.Control.Current_Alarm,eu:=VFD.Data.Motor_Current,Debounce_Active:=FALSE,status=>VFD.Control.Current_Status.eStatus);
lclAlarm_Active.SET:=FALSE;
IF Current_Alarm_EN THEN
	CASE Alarm.Status OF
		Burkert.eSensor_Status.HiHi_Alarm:
			VFD.Status.eStatus:=eVFD_Status.High_High_Current_Alarm;
			lclStatus:=VFD.Status.eStatus;
			lclAlarm_Active.SET:=TRUE;
		Burkert.eSensor_Status.High_Warning:
			VFD.Status.eStatus:=eVFD_Status.High_Current_Warning;
			//lclStatus:=VFD.Status.eStatus;
			//lclAlarm_Active.SET:=TRUE;
		Burkert.eSensor_Status.Low_Warning:
			VFD.Status.eStatus:=eVFD_Status.Low_Current_Warning;
			//lclStatus:=VFD.Status.eStatus;
			//lclAlarm_Active.SET:=TRUE;
		Burkert.eSensor_Status.Low_Low_Alarm:
			VFD.Status.eStatus:=eVFD_Status.Low_Low_Current_Alarm;
			lclStatus:=VFD.Status.eStatus;
			lclAlarm_Active.SET:=TRUE;
	END_CASE
END_IF;

IF VFD.Output_Pct>50 AND VFD.Data.Motor_Current<0.1 THEN
	VFD.Status.eStatus:=eVFD_Status.No_Motor_Load_Detected;
	lclStatus:=VFD.Status.eStatus;
	lclAlarm_Active.SET:=TRUE;
END_IF;

IF lclAlarm_Active.Q1 THEN
	VFD.Status.eStatus:=lclStatus;
	VFD_CMD_PCT:=0;
	VFD_Run:=FALSE;
END_IF;


T_1m(PT:=T#60S);
IF T_1m.Q AND VFD.Data.Drive_STATUS.Run THEN
	VFD.Control.RunTime_Minutes:=VFD.Control.RunTime_Minutes+1;
END_IF;


IF Max_hz >0 THEN	
	VFD.Output_Pct :=  (VFD.Output_Hz/ Max_hz)*100;//  VFD_CMD_PCT;
ELSE
	VFD.Output_Pct := VFD.Output_Hz;
END_IF;
END_ACTION

END_FUNCTION_BLOCK

// VFD_GS20_UDFB
FUNCTION_BLOCK VFD_GS20_UDFB
VAR_INPUT
	Interlock_NC:BOOL;
	Permissive_NC:BOOL;
	Connected:BOOL;
	VFD: REFERENCE TO cVFD_GS20_DUT;;
	Max_Hz:REAL;
END_VAR
VAR_OUTPUT
	//tx	:ARRAY[0..2] OF WORD;
	//tx2_send	:BOOL;
END_VAR
VAR
	vfd_cmd: REAL;
	PLC_RUN_WORD: WORD;
	TOF_0: TOF;
	SP: REAL;
	//VFD_CMD_PCT:REAL;
END_VAR

//VAR_IN_OUT
//	VFD	:	cVFD_GS20_DUT;
//END_VAR

(* body of a kind this reader does not render *)

ACTION Status:
VFD.Data.Drive_STATUS.Ready:=VFD.Data.STATUS2.1;
VFD.Data.Drive_STATUS.Run:=VFD.Data.STATUS2.0;
VFD.Data.Drive_STATUS.Fault:=VFD.Data.STATUS1>1 AND VFD.Data.STATUS1<255;

//VFD.Data.Drive_STATUS.






VFD.Ready:=(Connected AND VFD.MODE.eMode=eVFD_Modes.Auto AND VFD.Data.Drive_STATUS.Ready);
VFD.Status:=eVFD_Status.READY;
IF VFD.Data.Drive_STATUS.Run AND VFD.MODE.eMode=eVFD_Modes.Manual AND VFD.Data.Drive_STATUS.At_Speed THEN	VFD.Status:=eVFD_Status.M_Runing; END_IF;
IF VFD.Data.Drive_STATUS.Run AND VFD.MODE.eMode=eVFD_Modes.Auto AND VFD.Data.Drive_STATUS.At_Speed THEN VFD.Status:=eVFD_Status.A_Running; END_IF;

IF VFD.Data.Drive_STATUS.Run  AND NOT(VFD.Data.Drive_STATUS.At_Speed) THEN VFD.Status:=eVFD_Status.Ramping; END_IF;


IF VFD.MODE.eMode=eVFD_Modes.Auto AND NOT(Permissive_NC) THEN VFD.Status:=eVFD_Status.Interlocked; END_IF;





IF VFD.Data.Drive_STATUS.Fault THEN 
	VFD.Status:=eVFD_Status.Fault; 
	//VFD_CMD_PCT:=0;
	//VFD_Run:=FALSE;
END_IF;
IF VFD.MODE.eMode=eVFD_Modes.Disabled THEN VFD.Status:=eVFD_Status.Disabled; END_IF;
IF NOT(Interlock_NC) THEN 
		VFD.Status:=eVFD_Status.LOCKED_OUT; 
		//VFD_CMD_PCT:=0;
		//VFD_Run:=FALSE;
END_IF;
IF NOT(Connected) THEN 
	VFD.Status:=eVFD_Status.Offline;
	//VFD_CMD_PCT:=0;
	//VFD.Output_Pct:=0;
	//VFD_Run:=FALSE;
END_IF;
END_ACTION

END_FUNCTION_BLOCK

// VFD_GS2_UDFB
FUNCTION_BLOCK VFD_GS2_UDFB
VAR_INPUT
	rx	:ARRAY[0..11] OF WORD;
	Interlock:BOOL:=FALSE;
END_VAR
VAR_OUTPUT
	tx1	:ARRAY[0..2] OF WORD;
	tx2	:ARRAY[0..2] OF WORD;
END_VAR
VAR
	vfd_cmd: REAL;
	PLC_RUN_WORD: WORD;
	CTRL_PID_0: BURKERT_OSCAT_BASIC.CTRL_PID;
	PID_SP: REAL;
	PID_CV: REAL;
	TOF_0: TOF;
	PID_Enable: BOOL;
END_VAR

VAR_IN_OUT
	VFD_GS2_DUT	:	VFD_GS2_DUT;
	//Status:VFD_Status_DUT;
END_VAR
VAR // added by the converter: edge detectors and wires of the graphical bodies
    _w1 : BOOL;
END_VAR

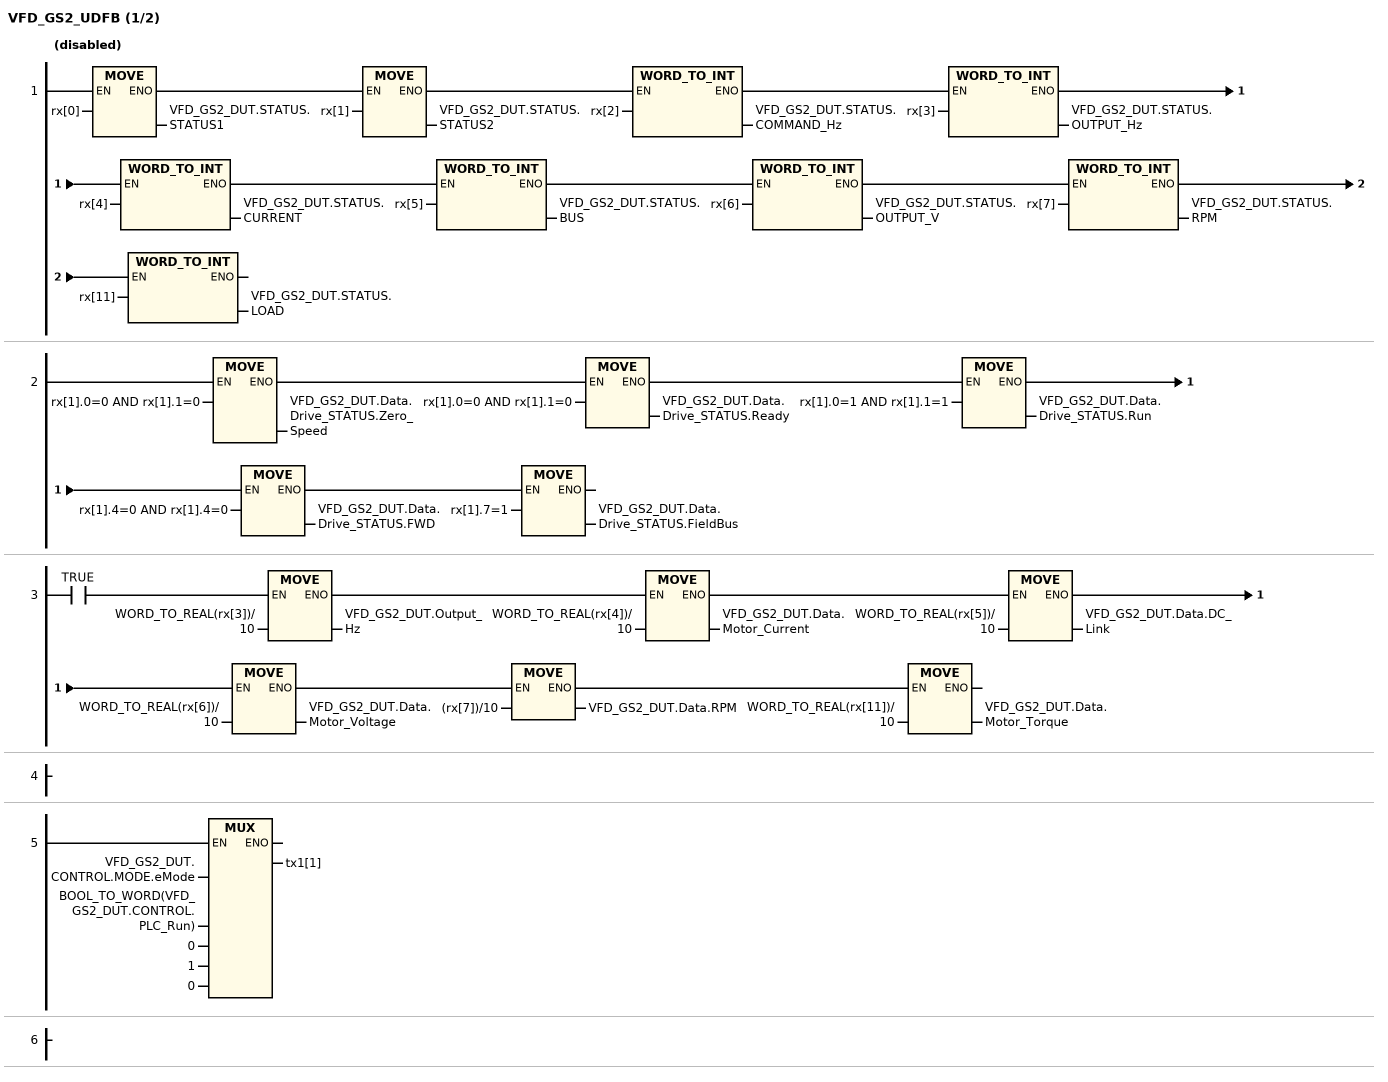
// NETWORK 1 (disabled)
// VFD_GS2_DUT.STATUS.STATUS1 := rx[0];
// VFD_GS2_DUT.STATUS.STATUS2 := rx[1];
// VFD_GS2_DUT.STATUS.COMMAND_Hz := WORD_TO_INT(rx[2]);
// VFD_GS2_DUT.STATUS.OUTPUT_Hz := WORD_TO_INT(rx[3]);
// VFD_GS2_DUT.STATUS.CURRENT := WORD_TO_INT(rx[4]);
// VFD_GS2_DUT.STATUS.BUS := WORD_TO_INT(rx[5]);
// VFD_GS2_DUT.STATUS.OUTPUT_V := WORD_TO_INT(rx[6]);
// VFD_GS2_DUT.STATUS.RPM := WORD_TO_INT(rx[7]);
// VFD_GS2_DUT.STATUS.LOAD := WORD_TO_INT(rx[11]);

// NETWORK 2
VFD_GS2_DUT.Data.Drive_STATUS.Zero_Speed := rx[1].0=0 AND rx[1].1=0;
VFD_GS2_DUT.Data.Drive_STATUS.Ready := rx[1].0=0 AND rx[1].1=0;
VFD_GS2_DUT.Data.Drive_STATUS.Run := rx[1].0=1 AND rx[1].1=1;
VFD_GS2_DUT.Data.Drive_STATUS.FWD := rx[1].4=0 AND rx[1].4=0;
VFD_GS2_DUT.Data.Drive_STATUS.FieldBus := rx[1].7=1;

// NETWORK 3
VFD_GS2_DUT.Output_Hz := WORD_TO_REAL(rx[3])/10;
VFD_GS2_DUT.Data.Motor_Current := WORD_TO_REAL(rx[4])/10;
VFD_GS2_DUT.Data.DC_Link := WORD_TO_REAL(rx[5])/10;
VFD_GS2_DUT.Data.Motor_Voltage := WORD_TO_REAL(rx[6])/10;
VFD_GS2_DUT.Data.RPM := (rx[7])/10;
VFD_GS2_DUT.Data.Motor_Torque := WORD_TO_REAL(rx[11])/10;

// NETWORK 4

// NETWORK 5
tx1[1] := MUX(VFD_GS2_DUT.CONTROL.MODE.eMode, BOOL_TO_WORD(VFD_GS2_DUT.CONTROL.PLC_Run), 0, 1, 0);

// NETWORK 6

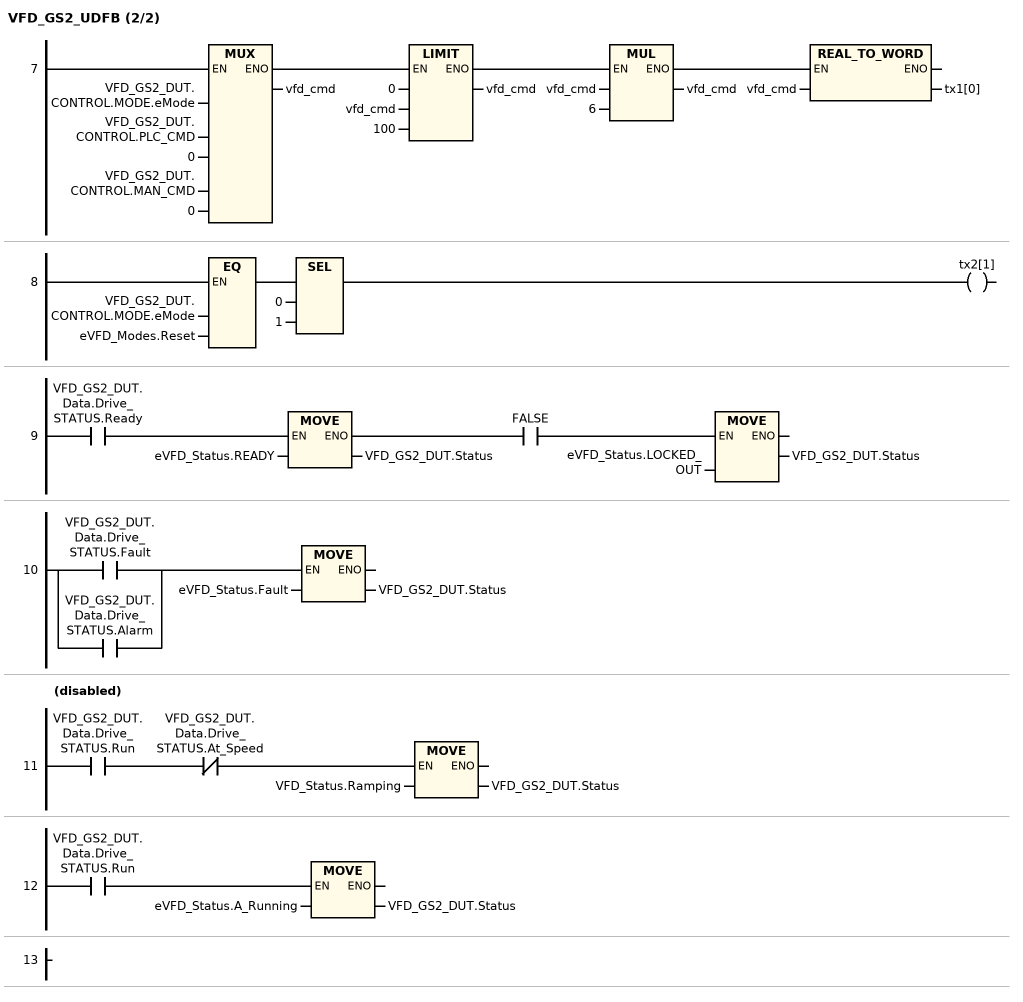
// NETWORK 7
vfd_cmd := MUX(VFD_GS2_DUT.CONTROL.MODE.eMode, VFD_GS2_DUT.CONTROL.PLC_CMD, 0, VFD_GS2_DUT.CONTROL.MAN_CMD, 0);
vfd_cmd := LIMIT(0, vfd_cmd, 100);
vfd_cmd := vfd_cmd * 6;
tx1[0] := REAL_TO_WORD(vfd_cmd);

// NETWORK 8
tx2[1] := SEL(VFD_GS2_DUT.CONTROL.MODE.eMode = eVFD_Modes.Reset, 0, 1);

// NETWORK 9
_w1 := VFD_GS2_DUT.Data.Drive_STATUS.Ready;
IF _w1 THEN VFD_GS2_DUT.Status := eVFD_Status.READY; END_IF
IF _w1 AND FALSE THEN VFD_GS2_DUT.Status := eVFD_Status.LOCKED_OUT; END_IF

// NETWORK 10
IF VFD_GS2_DUT.Data.Drive_STATUS.Fault OR VFD_GS2_DUT.Data.Drive_STATUS.Alarm THEN
    VFD_GS2_DUT.Status := eVFD_Status.Fault;
END_IF

// NETWORK 11 (disabled)
// IF VFD_GS2_DUT.Data.Drive_STATUS.Run AND NOT VFD_GS2_DUT.Data.Drive_STATUS.At_Speed THEN
//     VFD_GS2_DUT.Status := VFD_Status.Ramping;
// END_IF

// NETWORK 12
IF VFD_GS2_DUT.Data.Drive_STATUS.Run THEN VFD_GS2_DUT.Status := eVFD_Status.A_Running; END_IF

// NETWORK 13

END_FUNCTION_BLOCK

// VFD_Vacon100_UDFB
FUNCTION_BLOCK VFD_Vacon100_UDFB
VAR_INPUT
	Interlock:BOOL:=FALSE;
	Allow_Reverse:BOOL:=FALSE;
	Online:BOOL:=TRUE;
	Max_Hz:REAL:=60;
END_VAR
VAR_OUTPUT
	
END_VAR
VAR
	vfd_cmd: REAL;
	PLC_RUN_WORD: WORD;
	lcl_Run_Command: BOOL;
END_VAR

VAR_IN_OUT
	VFD	:	cVFD_Vacon;
END_VAR

(* body of a kind this reader does not render *)

END_FUNCTION_BLOCK

// Wago_750_455
FUNCTION_BLOCK Wago_750_455
VAR_INPUT
	//Raw:	REAL;

	Alarm_Enable:BOOL:=TRUE;
	Latching:BOOL:=FALSE;
	Fault:BOOL:=FALSE;
	Online:BOOL:=TRUE;
	Raw:REAl;
END_VAR

VAR_OUTPUT
	//Status	:BYTE;
END_VAR
VAR_IN_OUT
AIT	:	Burkert.cAIT;
END_VAR

VAR
	hihi: BOOL;
	hi: BOOL;
	lolo: BOOL;
	LO: BOOL;
	Alarm_Debounce: TON;
	deboune_Time: TIME;
	Alarm_Active: BOOL;
	Alarm_Debounce_ET: TIME;
	Alarm: BOOL;
	ALARM_2_0: BURKERT_OSCAT_BASIC.ALARM_2;
	F_TRIG_0: F_Trig;
	TON_0: TON;
	tmpEU: REAL;
	//tmpEU1: REAL;
	tmpEU2: REAL;
END_VAR

VAR_TEMP
	EU_Range: REAL;
	Raw_Range: REAL;
	Corrected_Raw: REAL;
	Raw_Pct: REAL;
	EU_Scaled: REAL;
END_VAR
VAR // added by the converter: edge detectors and wires of the graphical bodies
    _w1, _w2, _w3, _w4 : BOOL;
END_VAR

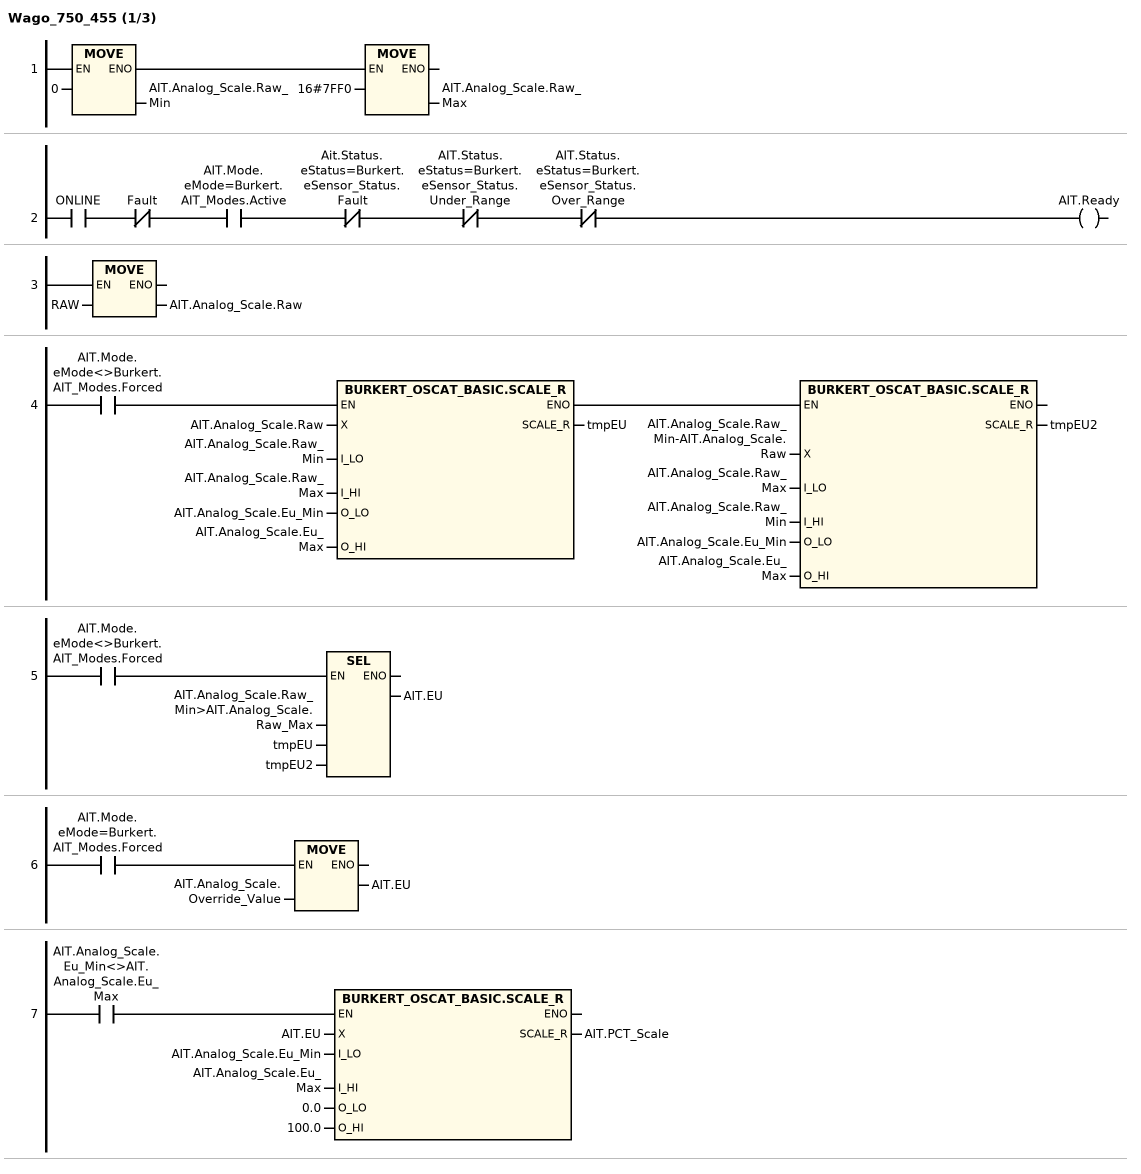
// NETWORK 1
AIT.Analog_Scale.Raw_Min := 0;
AIT.Analog_Scale.Raw_Max := 16#7FF0;

// NETWORK 2
AIT.Ready := ONLINE AND NOT Fault AND (AIT.Mode.eMode=Burkert.AIT_Modes.Active) AND NOT (Ait.Status.eStatus=Burkert.eSensor_Status.Fault) AND NOT (AIT.Status.eStatus=Burkert.eSensor_Status.Under_Range) AND NOT (AIT.Status.eStatus=Burkert.eSensor_Status.Over_Range);

// NETWORK 3
AIT.Analog_Scale.Raw := RAW;

// NETWORK 4
_w1 := AIT.Mode.eMode<>Burkert.AIT_Modes.Forced;
IF _w1 THEN
    tmpEU := BURKERT_OSCAT_BASIC.SCALE_R(X := AIT.Analog_Scale.Raw, I_LO := AIT.Analog_Scale.Raw_Min, I_HI := AIT.Analog_Scale.Raw_Max, O_LO := AIT.Analog_Scale.Eu_Min, O_HI := AIT.Analog_Scale.Eu_Max);
END_IF
IF _w1 THEN
    tmpEU2 := BURKERT_OSCAT_BASIC.SCALE_R(X := AIT.Analog_Scale.Raw_Min-AIT.Analog_Scale.Raw, I_LO := AIT.Analog_Scale.Raw_Max, I_HI := AIT.Analog_Scale.Raw_Min, O_LO := AIT.Analog_Scale.Eu_Min, O_HI := AIT.Analog_Scale.Eu_Max);
END_IF

// NETWORK 5
IF AIT.Mode.eMode<>Burkert.AIT_Modes.Forced THEN
    AIT.EU := SEL(AIT.Analog_Scale.Raw_Min>AIT.Analog_Scale.Raw_Max, tmpEU, tmpEU2);
END_IF

// NETWORK 6
IF AIT.Mode.eMode=Burkert.AIT_Modes.Forced THEN AIT.EU := AIT.Analog_Scale.Override_Value; END_IF

// NETWORK 7
IF AIT.Analog_Scale.Eu_Min<>AIT.Analog_Scale.Eu_Max THEN
    AIT.PCT_Scale := BURKERT_OSCAT_BASIC.SCALE_R(X := AIT.EU, I_LO := AIT.Analog_Scale.Eu_Min, I_HI := AIT.Analog_Scale.Eu_Max, O_LO := 0.0, O_HI := 100.0);
END_IF

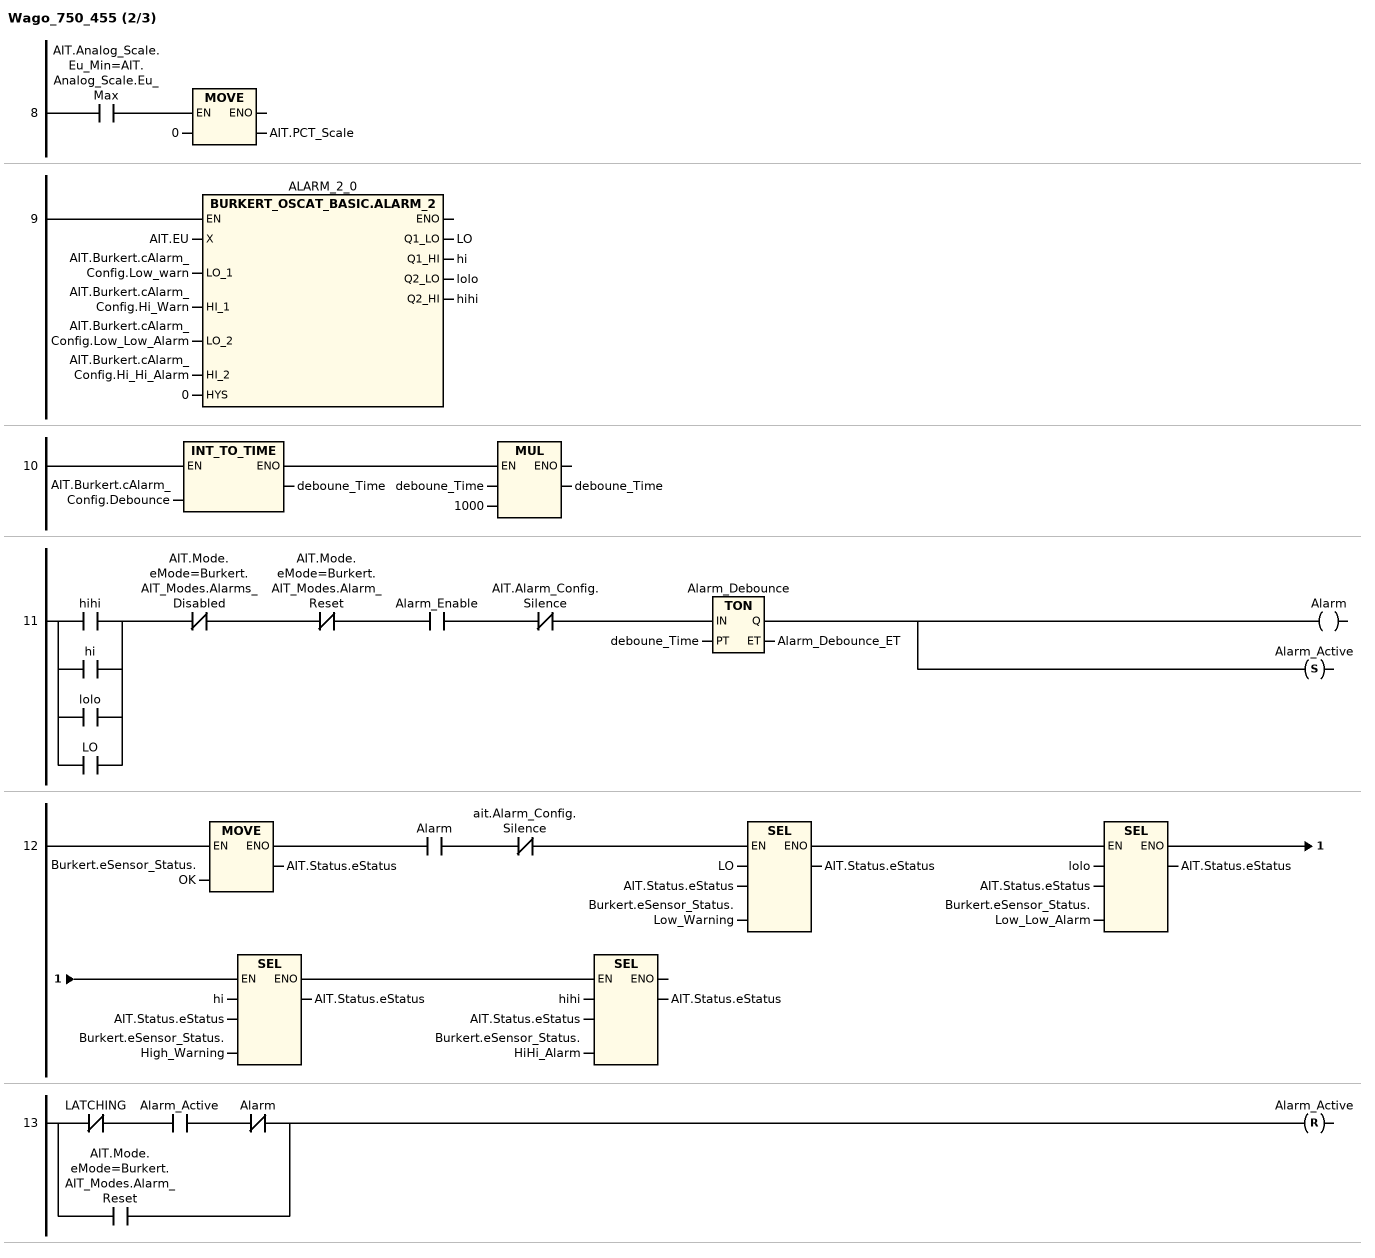
// NETWORK 8
IF AIT.Analog_Scale.Eu_Min=AIT.Analog_Scale.Eu_Max THEN AIT.PCT_Scale := 0; END_IF

// NETWORK 9
ALARM_2_0(
    X := AIT.EU,
    LO_1 := AIT.Burkert.cAlarm_Config.Low_warn,
    HI_1 := AIT.Burkert.cAlarm_Config.Hi_Warn,
    LO_2 := AIT.Burkert.cAlarm_Config.Low_Low_Alarm,
    HI_2 := AIT.Burkert.cAlarm_Config.Hi_Hi_Alarm,
    HYS := 0,
    Q1_LO => LO,
    Q1_HI => hi,
    Q2_LO => lolo,
    Q2_HI => hihi); // BURKERT_OSCAT_BASIC.ALARM_2

// NETWORK 10
deboune_Time := INT_TO_TIME(AIT.Burkert.cAlarm_Config.Debounce);
deboune_Time := deboune_Time * 1000;

// NETWORK 11
Alarm_Debounce(
    IN := (hihi OR hi OR lolo OR LO) AND NOT (AIT.Mode.eMode=Burkert.AIT_Modes.Alarms_Disabled) AND NOT (AIT.Mode.eMode=Burkert.AIT_Modes.Alarm_Reset) AND Alarm_Enable AND NOT AIT.Alarm_Config.Silence,
    PT := deboune_Time,
    ET => Alarm_Debounce_ET); // TON
Alarm := Alarm_Debounce.Q;
Alarm_Active S= Alarm_Debounce.Q;

// NETWORK 12
AIT.Status.eStatus := Burkert.eSensor_Status.OK;
_w2 := Alarm AND NOT ait.Alarm_Config.Silence;
IF _w2 THEN AIT.Status.eStatus := SEL(LO, AIT.Status.eStatus, Burkert.eSensor_Status.Low_Warning); END_IF
IF _w2 THEN AIT.Status.eStatus := SEL(lolo, AIT.Status.eStatus, Burkert.eSensor_Status.Low_Low_Alarm); END_IF
IF _w2 THEN AIT.Status.eStatus := SEL(hi, AIT.Status.eStatus, Burkert.eSensor_Status.High_Warning); END_IF
IF _w2 THEN AIT.Status.eStatus := SEL(hihi, AIT.Status.eStatus, Burkert.eSensor_Status.HiHi_Alarm); END_IF

// NETWORK 13
Alarm_Active R= NOT LATCHING AND Alarm_Active AND NOT Alarm OR (AIT.Mode.eMode=Burkert.AIT_Modes.Alarm_Reset);

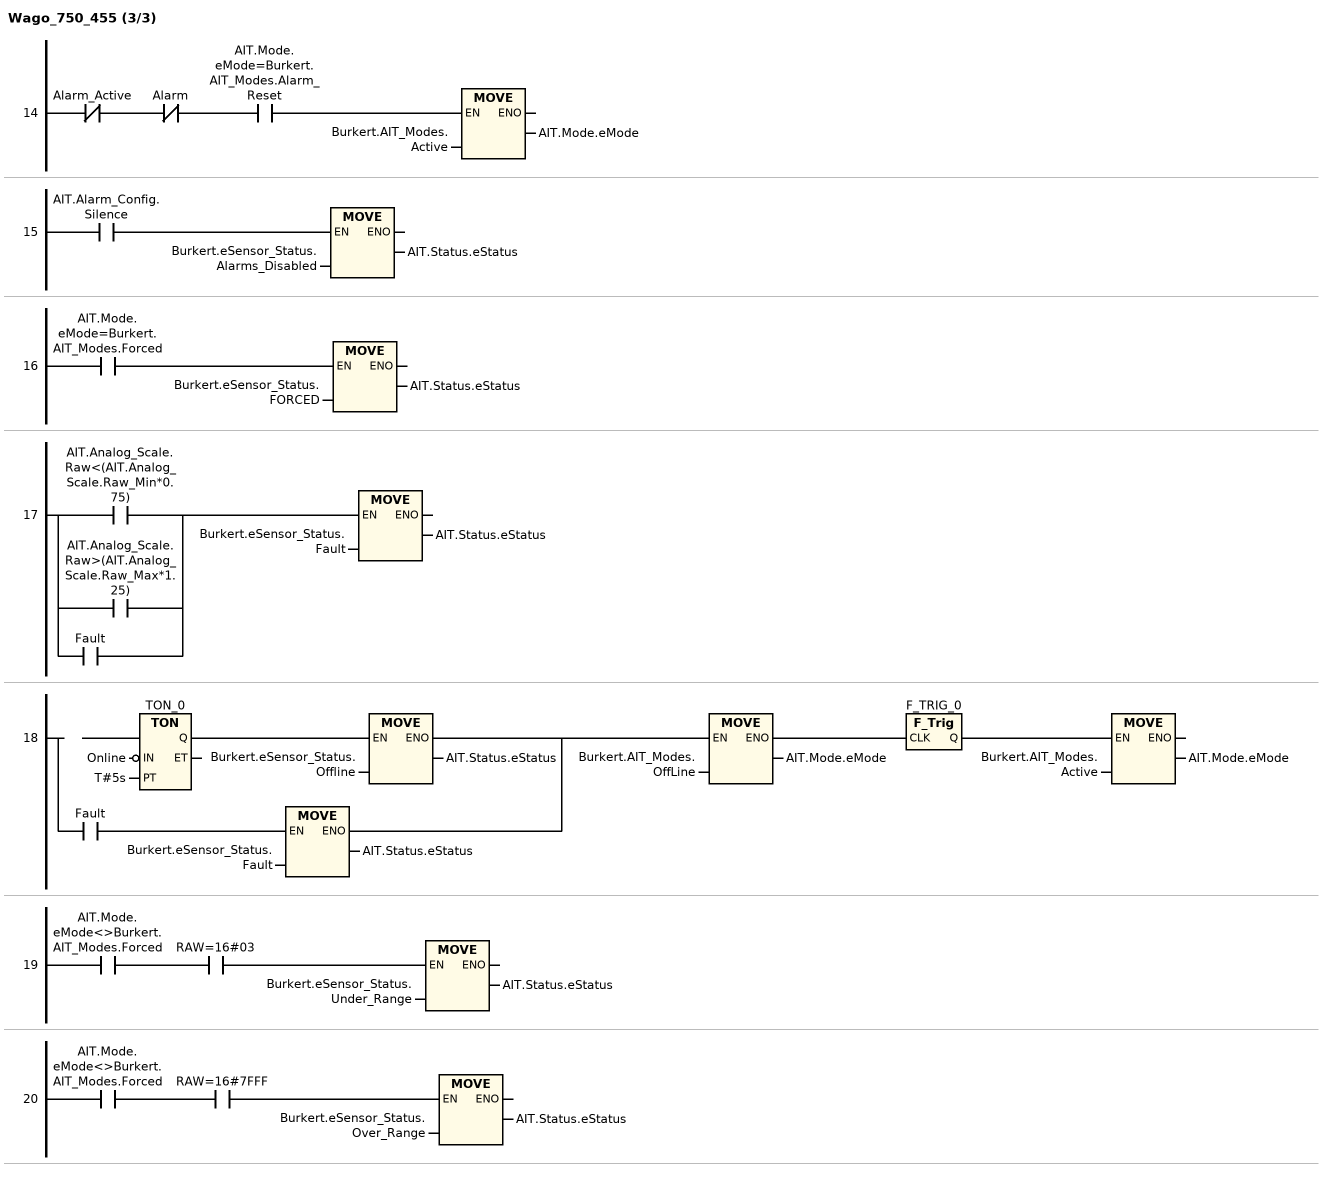
// NETWORK 14
IF NOT Alarm_Active AND NOT Alarm AND (AIT.Mode.eMode=Burkert.AIT_Modes.Alarm_Reset) THEN
    AIT.Mode.eMode := Burkert.AIT_Modes.Active;
END_IF

// NETWORK 15
IF AIT.Alarm_Config.Silence THEN AIT.Status.eStatus := Burkert.eSensor_Status.Alarms_Disabled; END_IF

// NETWORK 16
IF AIT.Mode.eMode=Burkert.AIT_Modes.Forced THEN AIT.Status.eStatus := Burkert.eSensor_Status.FORCED; END_IF

// NETWORK 17
IF (AIT.Analog_Scale.Raw<(AIT.Analog_Scale.Raw_Min*0.75)) OR (AIT.Analog_Scale.Raw>(AIT.Analog_Scale.Raw_Max*1.25)) OR Fault THEN
    AIT.Status.eStatus := Burkert.eSensor_Status.Fault;
END_IF

// NETWORK 18
TON_0(IN := NOT Online, PT := T#5s); // TON
_w3 := TON_0.Q;
IF _w3 THEN AIT.Status.eStatus := Burkert.eSensor_Status.Offline; END_IF
_w4 := Fault;
IF _w4 THEN AIT.Status.eStatus := Burkert.eSensor_Status.Fault; END_IF
IF _w3 OR _w4 THEN AIT.Mode.eMode := Burkert.AIT_Modes.OffLine; END_IF
F_TRIG_0(CLK := _w3 OR _w4); // F_Trig
IF F_TRIG_0.Q THEN AIT.Mode.eMode := Burkert.AIT_Modes.Active; END_IF

// NETWORK 19
IF (AIT.Mode.eMode<>Burkert.AIT_Modes.Forced) AND (RAW=16#03) THEN
    AIT.Status.eStatus := Burkert.eSensor_Status.Under_Range;
END_IF

// NETWORK 20
IF (AIT.Mode.eMode<>Burkert.AIT_Modes.Forced) AND (RAW=16#7FFF) THEN
    AIT.Status.eStatus := Burkert.eSensor_Status.Over_Range;
END_IF

END_FUNCTION_BLOCK

// Wago_750_NAMUR_NE43
FUNCTION_BLOCK Wago_750_NAMUR_NE43// EXTENDS Analog_Alarm_UDFB
VAR_INPUT
	Alarm_Enable:BOOL:=TRUE;
	Latching:BOOL:=FALSE;
	Fault:BOOL:=FALSE;
	Online:BOOL:=TRUE;
	//Raw:WORD;
END_VAR

VAR_OUTPUT
	//tInt:INT;
END_VAR
VAR_IN_OUT
AIT	:	Burkert.cAIT;
END_VAR

VAR
	//hihi: BOOL;
///	hi: BOOL;
	//lolo: BOOL;
	//LO: BOOL;
	//Alarm_Debounce: TON;
	//deboune_Time: TIME;
	//Alarm_Active: BOOL;
	//Alarm_Debounce_ET: TIME;
	//Alarm: BOOL;
	//ALARM_2_0: BURKERT_OSCAT_BASIC.ALARM_2;
	F_TRIG_0: F_Trig;
	TON_0: TON;
	tmpEU: REAL;
	tmpEU2: REAL;
	Alarm: Burkert.Analog_Alarm_UDFB;
END_VAR

VAR_TEMP
	tRaw:REAL;
	EU_ma:REAL;
END_VAR


(*
20.5 ma = 31800
3.8 ma = -392

Range is 32192 over 16.7 ma	  1927.66467 Counts ma
3.6 =  770.8 / -765
	3.8 =  0-(385)
	4 ma = 0
	12 ma = 15416 ( 1927 /ma
	20 ma =  30832 (1927/ ma
	20.5 ma = 31800 Doc
21 ma = 32759
0.1 ma =  192.7


*)

(* body of a kind this reader does not render *)

END_FUNCTION_BLOCK

// Burkert Library/ASi/ASi_8694_HMI_Sync_UDFB
FUNCTION_BLOCK ASi_8694_HMI_Sync_UDFB
VAR_INPUT
	Sync:BOOL;
END_VAR
VAR_OUTPUT
END_VAR
VAR
	Buffer:Burkert.ASi_8694;
	R_Trig_0: R_trig;
	Sync_1: BOOL;
	Sync_2: BOOL;
	PLC_Changes:UINT;
	HMI_Changes:UINT;
	
END_VAR

VAR_IN_OUT
	HMI:Burkert.ASi_8694;
	Local:Burkert.ASi_8694;
END_VAR

(* body of a kind this reader does not render *)

END_FUNCTION_BLOCK

// Burkert Library/Level_1/ACV_HMI_Sync_UDFB
FUNCTION_BLOCK ACV_HMI_Sync_UDFB
VAR_INPUT
	Sync:BOOL;
END_VAR
VAR_OUTPUT
	strMode:STRING;
	strStatus:STRING;
END_VAR
VAR
	Buffer:Burkert.cACV;
	R_Trig_0: R_trig;
	Sync_1: BOOL;
	Sync_2: BOOL;
	PLC_Changes:UINT;
	HMI_Changes:UINT;
	
	HMI_Change: BOOL;
END_VAR

VAR_IN_OUT
	HMI:Burkert.cACV;
	Local:Burkert.cACV;
END_VAR

(* body of a kind this reader does not render *)

END_FUNCTION_BLOCK

// Burkert Library/Level_1/AIT_HMI_Sync_UDFB
FUNCTION_BLOCK AIT_HMI_Sync_UDFB
VAR_INPUT
	Sync:BOOL;
END_VAR
VAR_OUTPUT
	strMode:STRING;
	strStatus:STRING;
END_VAR
VAR
	Buffer:Burkert.cAIT;
	R_Trig_0: R_trig;
	Sync_1: BOOL;
	Sync_2: BOOL;
	PLC_Changes:UINT;
	HMI_Changes:UINT;
	
END_VAR

VAR_IN_OUT
	HMI:Burkert.cAIT;
	Local:Burkert.cAIT;
END_VAR

(* body of a kind this reader does not render *)

END_FUNCTION_BLOCK

// Burkert Library/Level_1/B8050_HMI_Sync_UDFB
FUNCTION_BLOCK B8050_HMI_Sync_UDFB
VAR_INPUT
	Sync:BOOL;
END_VAR
VAR_OUTPUT
END_VAR
VAR
	R_Trig_0: R_trig;
	Buffer_HMI_reset:BOOL;
END_VAR

VAR_IN_OUT
	HMI:c8050;
	Local:c8050;
END_VAR

(* body of a kind this reader does not render *)

END_FUNCTION_BLOCK

// Burkert Library/Level_1/BCV_HMI_Sync_UDFB
FUNCTION_BLOCK BCV_HMI_Sync_UDFB
VAR_INPUT
	Sync:BOOL;
END_VAR
VAR_OUTPUT
	strMode:STRING;
	strStatus:STRING;
END_VAR
VAR
	Buffer:Burkert.cBCV;
	R_Trig_0: R_trig;
	Sync_1: BOOL;
	Sync_2: BOOL;
	PLC_Changes:UINT;
	HMI_Changes:UINT;
	
END_VAR

VAR_IN_OUT
	HMI:Burkert.cBCV;
	Local:Burkert.cBCV;
END_VAR

(* body of a kind this reader does not render *)

END_FUNCTION_BLOCK

// Burkert Library/Level_1/c8691_HMI_Sync_UDFB
FUNCTION_BLOCK c8691_HMI_Sync_UDFB
VAR_INPUT
	Sync:BOOL;
END_VAR
VAR_OUTPUT
	strMode:STRING;
	strStatus:STRING;
END_VAR
VAR
	Buffer:c8691;
	R_Trig_0: R_trig;
	Sync_1: BOOL;
	Sync_2: BOOL;
	PLC_Changes:UINT;
	HMI_Changes:UINT;
	
END_VAR

VAR_IN_OUT
	HMI:c8691;
	Local:c8691;
END_VAR

(* body of a kind this reader does not render *)

END_FUNCTION_BLOCK

// Burkert Library/Level_1/c8694_HMI_Sync_UDFB
FUNCTION_BLOCK c8694_HMI_Sync_UDFB
VAR_INPUT
	Sync:BOOL;
END_VAR
VAR_OUTPUT
	strMode:STRING;
	strStatus:STRING;
END_VAR
VAR
	Buffer:c8694;
	R_Trig_0: R_trig;
	Sync_1: BOOL;
	Sync_2: BOOL;
	PLC_Changes:UINT;
	HMI_Changes:UINT;
	
	HMI_Change: BOOL;
END_VAR

VAR_IN_OUT
	HMI:c8694;
	Local:c8694;
END_VAR

(* body of a kind this reader does not render *)

END_FUNCTION_BLOCK

// Burkert Library/Level_1/DI_HMI_Sync_UDFB
FUNCTION_BLOCK DI_HMI_Sync_UDFB
VAR_INPUT
	Sync:BOOL;
END_VAR
VAR_OUTPUT
	strMode:STRING;
	strStatus:STRING;
END_VAR
VAR
	Buffer:Burkert.DI_DUT;
	R_Trig_0: R_trig;
	Sync_1: BOOL;
	Sync_2: BOOL;
	PLC_Changes:UINT;
	HMI_Changes:UINT;
	
END_VAR

VAR_IN_OUT
	HMI:Burkert.DI_DUT;
	Local:Burkert.DI_DUT;
END_VAR

(* body of a kind this reader does not render *)

END_FUNCTION_BLOCK

// Burkert Library/Level_1/FIT_HMI_Sync_UDFB
FUNCTION_BLOCK FIT_HMI_Sync_UDFB
VAR_INPUT
	Sync:BOOL;
END_VAR
VAR_OUTPUT
	strMode:STRING;
	StrStatus:STRING;
END_VAR
VAR
	Buffer:Burkert.cFIT;
	R_Trig_0: R_trig;
	Sync_1: BOOL;
	Sync_2: BOOL;
	PLC_Changes:UINT;
	HMI_Changes:UINT;
	
END_VAR

VAR_IN_OUT
	HMI:Burkert.cFIT;
	Local:Burkert.cFIT;
END_VAR

(* body of a kind this reader does not render *)

END_FUNCTION_BLOCK

// Burkert Library/Level_1/GS20_VFD_HMI_Sync
FUNCTION_BLOCK GS20_VFD_HMI_Sync
VAR_INPUT
	Sync:BOOL;
END_VAR
VAR_OUTPUT
	StrStatus:STRING;
	StrMode:String;
END_VAR
VAR
	Buffer:cVFD_GS20_DUT;
	R_Trig_0: R_trig;
	Sync_1: BOOL;
	Sync_2: BOOL;
	PLC_Changes:UINT;
	HMI_Changes:UINT;
	
END_VAR

VAR_IN_OUT
	HMI:cVFD_GS20_DUT;
	Local:cVFD_GS20_DUT;
END_VAR

(* body of a kind this reader does not render *)

END_FUNCTION_BLOCK

// Burkert Library/Level_1/s336x_HMI_Sync
FUNCTION_BLOCK s336x_HMI_Sync
VAR_INPUT
	Sync:BOOL;
END_VAR
VAR_OUTPUT
	strMode:STRING;
	strStatus:STRING;
	StrNamurNe107:STRING;
END_VAR
VAR
	Buffer:c336x;
	R_Trig_0: R_trig;
	Sync_1: BOOL;
	Sync_2: BOOL;
	PLC_Changes:UINT;
	HMI_Changes:UINT;
	
	HMI_Change: BOOL;
END_VAR

VAR_IN_OUT
	HMI:c336x;
	Local:c336x;
END_VAR

(* body of a kind this reader does not render *)

END_FUNCTION_BLOCK

// Burkert Library/Level_1/s8050_HMI_Sync
FUNCTION_BLOCK s8050_HMI_Sync
VAR_INPUT
	Sync:BOOL;
END_VAR
VAR_OUTPUT
	strMode:STRING;
	strStatus:STRING;
END_VAR
VAR
	Buffer:c8050;
	R_Trig_0: R_trig;
	Sync_1: BOOL;
	Sync_2: BOOL;
	PLC_Changes:UINT;
	HMI_Changes:UINT;
	
END_VAR

VAR_IN_OUT
	HMI:c8050;
	Local:c8050;
END_VAR

(* body of a kind this reader does not render *)

END_FUNCTION_BLOCK

// Burkert Library/Level_1/s8098_HMI_Sync_UDFB
FUNCTION_BLOCK s8098_HMI_Sync_UDFB
VAR_INPUT
	Sync:BOOL;
END_VAR
VAR_OUTPUT
	//strMode:STRING;
	strNamur:STRING;
END_VAR
VAR
	Buffer:Burkert.c8098;
	R_Trig_0: R_trig;
	Sync_1: BOOL;
	Sync_2: BOOL;
	PLC_Changes:UINT;
	HMI_Changes:UINT;
	
END_VAR

VAR_IN_OUT
	HMI:Burkert.c8098;
	Local:Burkert.c8098;
END_VAR

VAR_OUTPUT
	//Name:String;
END_VAR

(* body of a kind this reader does not render *)

END_FUNCTION_BLOCK

// Burkert Library/Level_1/s8312_HMI_Sync
FUNCTION_BLOCK s8312_HMI_Sync
VAR_INPUT
	Sync:BOOL;
END_VAR
VAR_OUTPUT
	strMode:STRING;
	strStatus:STRING;
END_VAR
VAR
	Buffer:c8312;
	R_Trig_0: R_trig;
	Sync_1: BOOL;
	Sync_2: BOOL;
	PLC_Changes:UINT;
	HMI_Changes:UINT;
	
END_VAR

VAR_IN_OUT
	HMI:c8312;
	Local:c8312;
END_VAR

(* body of a kind this reader does not render *)

END_FUNCTION_BLOCK

// Burkert Library/Level_1/SV_HMI_Sync
FUNCTION_BLOCK SV_HMI_Sync
VAR_INPUT
	Sync:BOOL;
END_VAR
VAR_OUTPUT
	strMode:STRING;
	strStatus:STRING;
END_VAR
VAR
	Buffer:SV_DUT;
	R_Trig_0: R_trig;
	Sync_1: BOOL;
	Sync_2: BOOL;
	PLC_Changes:UINT;
	HMI_Changes:UINT;
	
END_VAR

VAR_IN_OUT
	HMI:SV_DUT;
	Local:SV_DUT;
END_VAR

(* body of a kind this reader does not render *)

END_FUNCTION_BLOCK

// Burkert Library/Level_1/Vacon_HMI_Sync_UDFB
FUNCTION_BLOCK Vacon_HMI_Sync_UDFB
VAR_INPUT
	Sync:BOOL;
END_VAR
VAR_OUTPUT
END_VAR
VAR
	Buffer:VFD_Vacon_DUT;
	R_Trig_0: R_trig;
	Sync_1: BOOL;
	Sync_2: BOOL;
	PLC_Changes:UINT;
	HMI_Changes:UINT;
	
END_VAR

VAR_IN_OUT
	HMI:VFD_Vacon_DUT;
	Local:VFD_Vacon_DUT;
END_VAR

(* body of a kind this reader does not render *)

END_FUNCTION_BLOCK

// Level_1_Devices/Burkert Library/CanOpen/CanOpen_8098
FUNCTION_BLOCK CanOpen_8098
VAR_INPUT
	CanOpen:	REFERENCE TO _3SCOS.CANRemoteDevice_Diag;
	Temperature_Units:eUnits:=eUnits.C;
	Flow_Units:eUnits:=eUnits.lpm;
	Volume_Units:eUnits:=eUnits.l;
	
	
END_VAR
VAR_OUTPUT

END_VAR
VAR_IN_OUT
	Device:cCanOpen_8098;
END_VAR
VAR
	Status_CLK:Burkert_OSCAT_BASIC.CLK_PRG;
	SDO_CLK:Burkert_OSCAT_BASIC.CLK_PRG;
	AutoRead_CLK:Burkert_OSCAT_BASIC.CLK_PRG;
	SDO_Read:CIA405.SDO_READ4;
	SDO_Write:CIA405.SDO_WRITE_DATA;
	Write_Data:Bytes_Dword;
	GetState:CIA405.GET_STATE;
	
	Alarm:ARRAY[0..5] OF Burkert.Analog_Alarm_UDFB;
	
	HMI_Reset_Ton:TON;
	tReset_1 :BOOL;
	tReset_2 :BOOL;
	tMass_Reset_1:BOOL; 
	tMass_Reset_2:BOOL;
	
	R_Trig_Reset:ARRAY[0..3] OF R_Trig;
	
	
END_VAR
VAR // added by the converter: edge detectors and wires of the graphical bodies
    _w1, _w2, _w3, _w4, _w5 : BOOL;
END_VAR

